// TwinCAT 3 PLC project SSP_M
// ProgramVersion: 3.1.4024.0
// libraries:
//   EfficientIO Communicator, * (EfficientIO)
//   EfficientIO Energy Basic, * (EfficientIO)
//   EfficientIO ModbusTCP, * (EfficientIO)
//   Lynus Persistent Data V1, * (Lynus AG)
//   Lynus Standards, * (EfficientIO)
//   Tc2_EtherCAT, * (Beckhoff Automation GmbH)
//   Tc2_Standard, * (Beckhoff Automation GmbH)
//   Tc2_System, * (Beckhoff Automation GmbH)
//   Tc2_Utilities, * (Beckhoff Automation GmbH)
//   Tc3_Module, * (Beckhoff Automation GmbH)
// project tree:
//   / FastTask.TcTTO, PlcTask.TcTTO, SlowTask.TcTTO (not stored)
//   FBs/EL3443_DPM/DUTs/ E_EL3443_DPM_Phase.TcDUT (not stored), E_EL3443_DPM_Total.TcDUT (not stored), MDP5001_341_7CD731EE.TcDUT (not stored), MDP5001_341_I_7CD731EE.TcDUT (not stored), MDP5001_341_O_7CD731EE.TcDUT (not stored), ST_EL3443_DPM_MUX_REAL.TcDUT (not stored), ST_EL3443_DPM_MUX_ULINT.TcDUT (not stored), ST_EL3443_DPM_StatusLx.TcDUT (not stored), ST_EL3443_DPM_StatusTotal.TcDUT (not stored), ST_EL3443_DPM_VariantLx.TcDUT (not stored), ST_EL3443_DPM_VariantTotal.TcDUT (not stored), ST_EL3443_DPM_VariantValues.TcDUT (not stored)
//   FBs/EL3443_DPM/ FB_EL3443_DPM.TcPOU (not stored)
//   FBs/EL3446 FW02 or higher/DUTs/ E_EL3446_Phase.TcDUT (not stored), MDP5001_342_066CA8C6.TcDUT (not stored), MDP5001_342_I_066CA8C6.TcDUT (not stored), MDP5001_342_O_066CA8C6.TcDUT, ST_EL3446_MUX_REAL.TcDUT (not stored), ST_EL3446_MUX_ULINT.TcDUT (not stored), ST_EL3446_StatusIx.TcDUT (not stored), ST_EL3446_VariantIx.TcDUT (not stored), ST_EL3446_VariantValues.TcDUT (not stored)
//   FBs/EL3446 FW02 or higher/ FB_EL3446.TcPOU (not stored)
//   FBs/ FB_CoE_EL3443.TcPOU (not stored), FB_CoE_EL3446.TcPOU (not stored), FB_EM_Beckhoff_EL3443.TcPOU (not stored), FB_EM_Beckhoff_EL3446.TcPOU (not stored)
//   POUs/ prgComEffIO.TcPOU, prgEM.TcPOU, prgEMS.TcPOU, prgHW.TcPOU, prgModbus.TcPOU, prgPersistent.TcPOU, prgRWEffIO.TcPOU (not stored), prgVarEffIO.TcPOU (not stored)
// real-time tasks:
//   TASK MiddleTask: cycle T#10ms, priority 20, ADS port 350
//   TASK FastTask: cycle T#5ms, priority 19, ADS port 351
//   TASK SlowTask: cycle T#20ms, priority 21, ADS port 352
// I/O:
//   DEVICE Device 1 (Beckhoff CCAT)
//   DEVICE Device 2 (EtherCAT), AmsNetId 5.146.126.209.3.1
//     Term 1 (EK1200) [EK1200-5000 EtherCAT Power supply (2A E-Bus)]
//       Term 6 (EL3443) [EL3443 3Ch. Power Measuring]
//       Term 2 (EL3443) [EL3443 3Ch. Power Measuring]
//       Term 3 (EL3446) [EL3446 6 Ch.DPM Current Measurement Terminal]
//       Term 4 (EL3446) [EL3446 6 Ch.DPM Current Measurement Terminal]
//       Term 5 (EL9011) [EL9011 End Terminal]
//   DEVICE Gerät 3 (RT-Ethernet Protocol), AmsNetId 5.146.126.209.4.1
//     BK9050 (BK9050-0000 192.168.1.235)
// variable links:
//   SSP-M/SSP-M Instance <-> Device 2 (EtherCAT)/Term 1 (EK1200)/Term 2 (EL3443)
//     PlcTask Inputs/prgHW.MDP5001_342_DPM_Data_Data_{1..20} <-> DPM Data/Data {1..20}  (20 links)
//     PlcTask Inputs/prgHW.MDP5001_342_L1_Basic_Current <-> L1 Basic/Current
//     PlcTask Inputs/prgHW.MDP5001_342_L2_Basic_Current <-> L2 Basic/Current
//     PlcTask Inputs/prgHW.MDP5001_342_L3_Basic_Current <-> L3 Basic/Current
//     PlcTask Inputs/prgHW.MDP5001_342_L1_Basic_Voltage <-> L1 Basic/Voltage
//     PlcTask Inputs/prgHW.MDP5001_342_L2_Basic_Voltage <-> L2 Basic/Voltage
//     PlcTask Inputs/prgHW.MDP5001_342_L3_Basic_Voltage <-> L3 Basic/Voltage
//     PlcTask Inputs/prgHW.MDP5001_342_L1_Power_Active_Power <-> L1 Power/Active Power
//     PlcTask Inputs/prgHW.MDP5001_342_L2_Power_Active_Power <-> L2 Power/Active Power
//     PlcTask Inputs/prgHW.MDP5001_342_L3_Power_Active_Power <-> L3 Power/Active Power
//     PlcTask Inputs/prgHW.MDP5001_342_L1_Power_Apparent_Power <-> L1 Power/Apparent Power
//     PlcTask Inputs/prgHW.MDP5001_342_L2_Power_Apparent_Power <-> L2 Power/Apparent Power
//     PlcTask Inputs/prgHW.MDP5001_342_L3_Power_Apparent_Power <-> L3 Power/Apparent Power
//     PlcTask Inputs/prgHW.MDP5001_342_L1_Power_Power_Factor <-> L1 Power/Power Factor
//     PlcTask Inputs/prgHW.MDP5001_342_L2_Power_Power_Factor <-> L2 Power/Power Factor
//     PlcTask Inputs/prgHW.MDP5001_342_L3_Power_Power_Factor <-> L3 Power/Power Factor
//     PlcTask Inputs/prgHW.MDP5001_342_L1_Power_Reactive_Power <-> L1 Power/Reactive Power
//     PlcTask Inputs/prgHW.MDP5001_342_L2_Power_Reactive_Power <-> L2 Power/Reactive Power
//     PlcTask Inputs/prgHW.MDP5001_342_L3_Power_Reactive_Power <-> L3 Power/Reactive Power
//     PlcTask Inputs/prgHW.MDP5001_342_L1_Status_Current_Guard_Error <-> L1 Status/Current Guard Error
//     PlcTask Inputs/prgHW.MDP5001_342_L2_Status_Current_Guard_Error <-> L2 Status/Current Guard Error
//     PlcTask Inputs/prgHW.MDP5001_342_L3_Status_Current_Guard_Error <-> L3 Status/Current Guard Error
//     PlcTask Inputs/prgHW.MDP5001_342_L1_Status_Current_Guard_Warning <-> L1 Status/Current Guard Warning
//     PlcTask Inputs/prgHW.MDP5001_342_L2_Status_Current_Guard_Warning <-> L2 Status/Current Guard Warning
//     PlcTask Inputs/prgHW.MDP5001_342_L3_Status_Current_Guard_Warning <-> L3 Status/Current Guard Warning
//     PlcTask Inputs/prgHW.MDP5001_342_L1_Status_Inaccurate_Current <-> L1 Status/Inaccurate Current
//     PlcTask Inputs/prgHW.MDP5001_342_L2_Status_Inaccurate_Current <-> L2 Status/Inaccurate Current
//     PlcTask Inputs/prgHW.MDP5001_342_L3_Status_Inaccurate_Current <-> L3 Status/Inaccurate Current
//     PlcTask Inputs/prgHW.MDP5001_342_L1_Status_Inaccurate_Voltage <-> L1 Status/Inaccurate Voltage
//     PlcTask Inputs/prgHW.MDP5001_342_L2_Status_Inaccurate_Voltage <-> L2 Status/Inaccurate Voltage
//     PlcTask Inputs/prgHW.MDP5001_342_L3_Status_Inaccurate_Voltage <-> L3 Status/Inaccurate Voltage
//     PlcTask Inputs/prgHW.MDP5001_342_L1_Status_Overcurrent <-> L1 Status/Overcurrent
//     PlcTask Inputs/prgHW.MDP5001_342_L2_Status_Overcurrent <-> L2 Status/Overcurrent
//     PlcTask Inputs/prgHW.MDP5001_342_L3_Status_Overcurrent <-> L3 Status/Overcurrent
//     PlcTask Inputs/prgHW.MDP5001_342_L1_Status_Overvoltage <-> L1 Status/Overvoltage
//     PlcTask Inputs/prgHW.MDP5001_342_L2_Status_Overvoltage <-> L2 Status/Overvoltage
//     PlcTask Inputs/prgHW.MDP5001_342_L3_Status_Overvoltage <-> L3 Status/Overvoltage
//     PlcTask Inputs/prgHW.MDP5001_342_L1_Status_TxPDO_Toggle <-> L1 Status/TxPDO Toggle
//     PlcTask Inputs/prgHW.MDP5001_342_L2_Status_TxPDO_Toggle <-> L2 Status/TxPDO Toggle
//     PlcTask Inputs/prgHW.MDP5001_342_L3_Status_TxPDO_Toggle <-> L3 Status/TxPDO Toggle
//     PlcTask Inputs/prgHW.MDP5001_342_L1_Status_Voltage_Guard_Error <-> L1 Status/Voltage Guard Error
//     PlcTask Inputs/prgHW.MDP5001_342_L2_Status_Voltage_Guard_Error <-> L2 Status/Voltage Guard Error
//     PlcTask Inputs/prgHW.MDP5001_342_L3_Status_Voltage_Guard_Error <-> L3 Status/Voltage Guard Error
//     PlcTask Inputs/prgHW.MDP5001_342_L1_Status_Voltage_Guard_Warning <-> L1 Status/Voltage Guard Warning
//     PlcTask Inputs/prgHW.MDP5001_342_L2_Status_Voltage_Guard_Warning <-> L2 Status/Voltage Guard Warning
//     PlcTask Inputs/prgHW.MDP5001_342_L3_Status_Voltage_Guard_Warning <-> L3 Status/Voltage Guard Warning
//     PlcTask Inputs/prgHW.MDP5001_342_L1_Status_Voltage_Sign_Bit <-> L1 Status/Voltage Sign Bit
//     PlcTask Inputs/prgHW.MDP5001_342_L2_Status_Voltage_Sign_Bit <-> L2 Status/Voltage Sign Bit
//     PlcTask Inputs/prgHW.MDP5001_342_L3_Status_Voltage_Sign_Bit <-> L3 Status/Voltage Sign Bit
//     PlcTask Inputs/prgHW.MDP5001_342_Total_Basic_Calculated_Neutral_Line_Current <-> Total Basic/Calculated Neutral Line Current
//     PlcTask Inputs/prgHW.MDP5001_342_Total_Basic_Frequency <-> Total Basic/Frequency
//     PlcTask Inputs/prgHW.MDP5001_342_Total_Basic_Power_Factor <-> Total Basic/Power Factor
//     PlcTask Inputs/prgHW.MDP5001_342_Total_Status_Active_Power_Guard_Error <-> Total Status/Active Power Guard Error
//     PlcTask Inputs/prgHW.MDP5001_342_Total_Status_Active_Power_Guard_Warning <-> Total Status/Active Power Guard Warning
//     PlcTask Inputs/prgHW.MDP5001_342_Total_Status_Apparent_Power_Guard_Error <-> Total Status/Apparent Power Guard Error
//     PlcTask Inputs/prgHW.MDP5001_342_Total_Status_Apparent_Power_Guard_Warning <-> Total Status/Apparent Power Guard Warning
//     PlcTask Inputs/prgHW.MDP5001_342_Total_Status_Frequency_Guard_Error <-> Total Status/Frequency Guard Error
//     PlcTask Inputs/prgHW.MDP5001_342_Total_Status_Frequency_Guard_Warning <-> Total Status/Frequency Guard Warning
//     PlcTask Inputs/prgHW.MDP5001_342_Total_Status_Grid_Direction <-> Total Status/Grid Direction
//     PlcTask Inputs/prgHW.MDP5001_342_Total_Status_Neutral_Current_Guard_Error <-> Total Status/Neutral Current Guard Error
//     PlcTask Inputs/prgHW.MDP5001_342_Total_Status_Neutral_Current_Guard_Warning <-> Total Status/Neutral Current Guard Warning
//     PlcTask Inputs/prgHW.MDP5001_342_Total_Status_Power_Quality_Factor <-> Total Status/Power Quality Factor
//     PlcTask Inputs/prgHW.MDP5001_342_Total_Status_Power_Quality_Guard_Error <-> Total Status/Power Quality Guard Error
//     PlcTask Inputs/prgHW.MDP5001_342_Total_Status_Power_Quality_Guard_Warning <-> Total Status/Power Quality Guard Warning
//     PlcTask Inputs/prgHW.MDP5001_342_Total_Status_System_State <-> Total Status/System State
//     PlcTask Inputs/prgHW.MDP5001_342_Total_Status_TxPDO_State <-> Total Status/TxPDO State
//     PlcTask Inputs/prgHW.MDP5001_342_Total_Status_TxPDO_Toggle <-> Total Status/TxPDO Toggle
//     PlcTask Inputs/prgHW.MDP5001_342_Total_Variant_Value_In_Index_1_REAL <-> Total Variant Value In/Index 1 REAL
//     PlcTask Inputs/prgHW.MDP5001_342_Total_Variant_Value_In_Index_2_REAL <-> Total Variant Value In/Index 2 REAL
//     PlcTask Inputs/prgHW.MDP5001_342_Total_Variant_Value_In_Index_3_REAL <-> Total Variant Value In/Index 3 REAL
//     PlcTask Inputs/prgHW.MDP5001_342_Total_Variant_Value_In_Index_4_ULINT <-> Total Variant Value In/Index 4 ULINT
//     PlcTask Inputs/prgHW.MDP5001_342_Total_Variant_Value_In_TxPDO_Toggle <-> Total Variant Value In/TxPDO Toggle
//     PlcTask Inputs/prgHW.MDP5001_342_Total_Variant_Value_In_Value_1_REAL <-> Total Variant Value In/Value 1 REAL
//     PlcTask Inputs/prgHW.MDP5001_342_Total_Variant_Value_In_Value_2_REAL <-> Total Variant Value In/Value 2 REAL
//     PlcTask Inputs/prgHW.MDP5001_342_Total_Variant_Value_In_Value_3_REAL <-> Total Variant Value In/Value 3 REAL
//     PlcTask Inputs/prgHW.MDP5001_342_Total_Variant_Value_In_Value_4_ULINT <-> Total Variant Value In/Value 4 ULINT
//     PlcTask Outputs/prgHW.MDP5001_342_Total_Interval_Reset_Interval <-> Total Interval/Reset Interval
//     PlcTask Outputs/prgHW.MDP5001_342_Total_Variant_Value_Out_Index_1_REAL <-> Total Variant Value Out/Index 1 REAL
//     PlcTask Outputs/prgHW.MDP5001_342_Total_Variant_Value_Out_Index_2_REAL <-> Total Variant Value Out/Index 2 REAL
//     PlcTask Outputs/prgHW.MDP5001_342_Total_Variant_Value_Out_Index_3_REAL <-> Total Variant Value Out/Index 3 REAL
//     PlcTask Outputs/prgHW.MDP5001_342_Total_Variant_Value_Out_Index_4_ULINT <-> Total Variant Value Out/Index 4 ULINT
//   SSP-M/SSP-M Instance <-> Device 2 (EtherCAT)/Term 1 (EK1200)/Term 3 (EL3446)
//     PlcTask Inputs/prgHW.MDP5001_342_DPM_Variant_Value_In_Index_1_REAL_1 <-> DPM Variant Value In/Index 1 REAL
//     PlcTask Inputs/prgHW.MDP5001_342_DPM_Variant_Value_In_Index_2_REAL_1 <-> DPM Variant Value In/Index 2 REAL
//     PlcTask Inputs/prgHW.MDP5001_342_DPM_Variant_Value_In_Index_3_REAL_1 <-> DPM Variant Value In/Index 3 REAL
//     PlcTask Inputs/prgHW.MDP5001_342_DPM_Variant_Value_In_Index_4_ULINT_1 <-> DPM Variant Value In/Index 4 ULINT
//     PlcTask Inputs/prgHW.MDP5001_342_DPM_Variant_Value_In_TxPDO_Toggle_1 <-> DPM Variant Value In/TxPDO Toggle
//     PlcTask Inputs/prgHW.MDP5001_342_DPM_Variant_Value_In_Value_1_REAL_1 <-> DPM Variant Value In/Value 1 REAL
//     PlcTask Inputs/prgHW.MDP5001_342_DPM_Variant_Value_In_Value_2_REAL_1 <-> DPM Variant Value In/Value 2 REAL
//     PlcTask Inputs/prgHW.MDP5001_342_DPM_Variant_Value_In_Value_3_REAL_1 <-> DPM Variant Value In/Value 3 REAL
//     PlcTask Inputs/prgHW.MDP5001_342_DPM_Variant_Value_In_Value_4_ULINT_1 <-> DPM Variant Value In/Value 4 ULINT
//     PlcTask Inputs/prgHW.MDP5001_342_I{1..6}_Channel_Active_Energy_1 <-> I{1..6} Channel/Active Energy  (6 links)
//     PlcTask Inputs/prgHW.MDP5001_342_I{1..6}_Channel_Active_Power_1 <-> I{1..6} Channel/Active Power  (6 links)
//     PlcTask Inputs/prgHW.MDP5001_342_I{1..6}_Channel_Active_Power_Guard_Error_1 <-> I{1..6} Channel/Active Power Guard Error  (6 links)
//     PlcTask Inputs/prgHW.MDP5001_342_I{1..6}_Channel_Active_Power_Guard_Warning_1 <-> I{1..6} Channel/Active Power Guard Warning  (6 links)
//     PlcTask Inputs/prgHW.MDP5001_342_I{1..6}_Channel_Apparent_Power_1 <-> I{1..6} Channel/Apparent Power  (6 links)
//     PlcTask Inputs/prgHW.MDP5001_342_I{1..6}_Channel_Apparent_Power_Guard_Error_1 <-> I{1..6} Channel/Apparent Power Guard Error  (6 links)
//     PlcTask Inputs/prgHW.MDP5001_342_I{1..6}_Channel_Apparent_Power_Guard_Warning_1 <-> I{1..6} Channel/Apparent Power Guard Warning  (6 links)
//     PlcTask Inputs/prgHW.MDP5001_342_I{1..6}_Channel_Current_1 <-> I{1..6} Channel/Current  (6 links)
//     PlcTask Inputs/prgHW.MDP5001_342_I{1..6}_Channel_Current_Guard_Error_1 <-> I{1..6} Channel/Current Guard Error  (6 links)
//     PlcTask Inputs/prgHW.MDP5001_342_I{1..6}_Channel_Current_Guard_Warning_1 <-> I{1..6} Channel/Current Guard Warning  (6 links)
//     PlcTask Inputs/prgHW.MDP5001_342_I{1..6}_Channel_DPM_Inaccurate_1 <-> I{1..6} Channel/DPM Inaccurate  (6 links)
//     PlcTask Inputs/prgHW.MDP5001_342_I{1..6}_Channel_DPM_Timeout_1 <-> I{1..6} Channel/DPM Timeout  (6 links)
//     PlcTask Inputs/prgHW.MDP5001_342_I{1..6}_Channel_Inaccurate_Current_1 <-> I{1..6} Channel/Inaccurate Current  (6 links)
//     PlcTask Inputs/prgHW.MDP5001_342_I{1..6}_Channel_Overcurrent_1 <-> I{1..6} Channel/Overcurrent  (6 links)
//     PlcTask Inputs/prgHW.MDP5001_342_I{1..6}_Channel_Reactive_Power_Fundamental_1 <-> I{1..6} Channel/Reactive Power Fundamental  (6 links)
//     PlcTask Inputs/prgHW.MDP5001_342_I{1..6}_Channel_Reactive_Power_Guard_Error_1 <-> I{1..6} Channel/Reactive Power Guard Error  (6 links)
//     PlcTask Inputs/prgHW.MDP5001_342_I{1..6}_Channel_Reactive_Power_Guard_Warning_1 <-> I{1..6} Channel/Reactive Power Guard Warning  (6 links)
//     PlcTask Inputs/prgHW.MDP5001_342_I{1..6}_Channel_TxPDO_Toggle_1 <-> I{1..6} Channel/TxPDO Toggle  (6 links)
//     PlcTask Outputs/prgHW.MDP5001_342_DPM_Data_Data_{1..20}_1 <-> DPM Data/Data {1..20}  (20 links)
//     PlcTask Outputs/prgHW.MDP5001_342_DPM_Variant_Value_Out_Index_1_REAL_1 <-> DPM Variant Value Out/Index 1 REAL
//     PlcTask Outputs/prgHW.MDP5001_342_DPM_Variant_Value_Out_Index_2_REAL_1 <-> DPM Variant Value Out/Index 2 REAL
//     PlcTask Outputs/prgHW.MDP5001_342_DPM_Variant_Value_Out_Index_3_REAL_1 <-> DPM Variant Value Out/Index 3 REAL
//     PlcTask Outputs/prgHW.MDP5001_342_DPM_Variant_Value_Out_Index_4_ULINT_1 <-> DPM Variant Value Out/Index 4 ULINT
//   SSP-M/SSP-M Instance <-> Device 2 (EtherCAT)/Term 1 (EK1200)/Term 4 (EL3446)
//     PlcTask Inputs/prgHW.MDP5001_342_DPM_Variant_Value_In_Index_1_REAL_2 <-> DPM Variant Value In/Index 1 REAL
//     PlcTask Inputs/prgHW.MDP5001_342_DPM_Variant_Value_In_Index_2_REAL_2 <-> DPM Variant Value In/Index 2 REAL
//     PlcTask Inputs/prgHW.MDP5001_342_DPM_Variant_Value_In_Index_3_REAL_2 <-> DPM Variant Value In/Index 3 REAL
//     PlcTask Inputs/prgHW.MDP5001_342_DPM_Variant_Value_In_Index_4_ULINT_2 <-> DPM Variant Value In/Index 4 ULINT
//     PlcTask Inputs/prgHW.MDP5001_342_DPM_Variant_Value_In_TxPDO_Toggle_2 <-> DPM Variant Value In/TxPDO Toggle
//     PlcTask Inputs/prgHW.MDP5001_342_DPM_Variant_Value_In_Value_1_REAL_2 <-> DPM Variant Value In/Value 1 REAL
//     PlcTask Inputs/prgHW.MDP5001_342_DPM_Variant_Value_In_Value_2_REAL_2 <-> DPM Variant Value In/Value 2 REAL
//     PlcTask Inputs/prgHW.MDP5001_342_DPM_Variant_Value_In_Value_3_REAL_2 <-> DPM Variant Value In/Value 3 REAL
//     PlcTask Inputs/prgHW.MDP5001_342_DPM_Variant_Value_In_Value_4_ULINT_2 <-> DPM Variant Value In/Value 4 ULINT
//     PlcTask Inputs/prgHW.MDP5001_342_I{1..6}_Channel_Active_Energy_2 <-> I{1..6} Channel/Active Energy  (6 links)
//     PlcTask Inputs/prgHW.MDP5001_342_I{1..6}_Channel_Active_Power_2 <-> I{1..6} Channel/Active Power  (6 links)
//     PlcTask Inputs/prgHW.MDP5001_342_I{1..6}_Channel_Active_Power_Guard_Error_2 <-> I{1..6} Channel/Active Power Guard Error  (6 links)
//     PlcTask Inputs/prgHW.MDP5001_342_I{1..6}_Channel_Active_Power_Guard_Warning_2 <-> I{1..6} Channel/Active Power Guard Warning  (6 links)
//     PlcTask Inputs/prgHW.MDP5001_342_I{1..6}_Channel_Apparent_Power_2 <-> I{1..6} Channel/Apparent Power  (6 links)
//     PlcTask Inputs/prgHW.MDP5001_342_I{1..6}_Channel_Apparent_Power_Guard_Error_2 <-> I{1..6} Channel/Apparent Power Guard Error  (6 links)
//     PlcTask Inputs/prgHW.MDP5001_342_I{1..6}_Channel_Apparent_Power_Guard_Warning_2 <-> I{1..6} Channel/Apparent Power Guard Warning  (6 links)
//     PlcTask Inputs/prgHW.MDP5001_342_I{1..6}_Channel_Current_2 <-> I{1..6} Channel/Current  (6 links)
//     PlcTask Inputs/prgHW.MDP5001_342_I{1..6}_Channel_Current_Guard_Error_2 <-> I{1..6} Channel/Current Guard Error  (6 links)
//     PlcTask Inputs/prgHW.MDP5001_342_I{1..6}_Channel_Current_Guard_Warning_2 <-> I{1..6} Channel/Current Guard Warning  (6 links)
//     PlcTask Inputs/prgHW.MDP5001_342_I{1..6}_Channel_DPM_Inaccurate_2 <-> I{1..6} Channel/DPM Inaccurate  (6 links)
//     PlcTask Inputs/prgHW.MDP5001_342_I{1..6}_Channel_DPM_Timeout_2 <-> I{1..6} Channel/DPM Timeout  (6 links)
//     PlcTask Inputs/prgHW.MDP5001_342_I{1..6}_Channel_Inaccurate_Current_2 <-> I{1..6} Channel/Inaccurate Current  (6 links)
//     PlcTask Inputs/prgHW.MDP5001_342_I{1..6}_Channel_Overcurrent_2 <-> I{1..6} Channel/Overcurrent  (6 links)
//     PlcTask Inputs/prgHW.MDP5001_342_I{1..6}_Channel_Reactive_Power_Fundamental_2 <-> I{1..6} Channel/Reactive Power Fundamental  (6 links)
//     PlcTask Inputs/prgHW.MDP5001_342_I{1..6}_Channel_Reactive_Power_Guard_Error_2 <-> I{1..6} Channel/Reactive Power Guard Error  (6 links)
//     PlcTask Inputs/prgHW.MDP5001_342_I{1..6}_Channel_Reactive_Power_Guard_Warning_2 <-> I{1..6} Channel/Reactive Power Guard Warning  (6 links)
//     PlcTask Inputs/prgHW.MDP5001_342_I{1..6}_Channel_TxPDO_Toggle_2 <-> I{1..6} Channel/TxPDO Toggle  (6 links)
//     PlcTask Outputs/prgHW.MDP5001_342_DPM_Data_Data_{1..20}_2 <-> DPM Data/Data {1..20}  (20 links)
//     PlcTask Outputs/prgHW.MDP5001_342_DPM_Variant_Value_Out_Index_1_REAL_2 <-> DPM Variant Value Out/Index 1 REAL
//     PlcTask Outputs/prgHW.MDP5001_342_DPM_Variant_Value_Out_Index_2_REAL_2 <-> DPM Variant Value Out/Index 2 REAL
//     PlcTask Outputs/prgHW.MDP5001_342_DPM_Variant_Value_Out_Index_3_REAL_2 <-> DPM Variant Value Out/Index 3 REAL
//     PlcTask Outputs/prgHW.MDP5001_342_DPM_Variant_Value_Out_Index_4_ULINT_2 <-> DPM Variant Value Out/Index 4 ULINT
//   SSP-M/SSP-M Instance <-> Device 2 (EtherCAT)/Term 1 (EK1200)/Term 6 (EL3443)
//     PlcTask Inputs/prgHW.MDP5001_341_DPM_Data_Data_{1..20} <-> DPM Data/Data {1..20}  (20 links)
//     PlcTask Inputs/prgHW.MDP5001_341_L1_Basic_Current <-> L1 Basic/Current
//     PlcTask Inputs/prgHW.MDP5001_341_L2_Basic_Current <-> L2 Basic/Current
//     PlcTask Inputs/prgHW.MDP5001_341_L3_Basic_Current <-> L3 Basic/Current
//     PlcTask Inputs/prgHW.MDP5001_341_L1_Basic_Voltage <-> L1 Basic/Voltage
//     PlcTask Inputs/prgHW.MDP5001_341_L2_Basic_Voltage <-> L2 Basic/Voltage
//     PlcTask Inputs/prgHW.MDP5001_341_L3_Basic_Voltage <-> L3 Basic/Voltage
//     PlcTask Inputs/prgHW.MDP5001_341_L1_Power_Active_Power <-> L1 Power/Active Power
//     PlcTask Inputs/prgHW.MDP5001_341_L2_Power_Active_Power <-> L2 Power/Active Power
//     PlcTask Inputs/prgHW.MDP5001_341_L3_Power_Active_Power <-> L3 Power/Active Power
//     PlcTask Inputs/prgHW.MDP5001_341_L1_Power_Apparent_Power <-> L1 Power/Apparent Power
//     PlcTask Inputs/prgHW.MDP5001_341_L2_Power_Apparent_Power <-> L2 Power/Apparent Power
//     PlcTask Inputs/prgHW.MDP5001_341_L3_Power_Apparent_Power <-> L3 Power/Apparent Power
//     PlcTask Inputs/prgHW.MDP5001_341_L1_Power_Power_Factor <-> L1 Power/Power Factor
//     PlcTask Inputs/prgHW.MDP5001_341_L2_Power_Power_Factor <-> L2 Power/Power Factor
//     PlcTask Inputs/prgHW.MDP5001_341_L3_Power_Power_Factor <-> L3 Power/Power Factor
//     PlcTask Inputs/prgHW.MDP5001_341_L1_Power_Reactive_Power <-> L1 Power/Reactive Power
//     PlcTask Inputs/prgHW.MDP5001_341_L2_Power_Reactive_Power <-> L2 Power/Reactive Power
//     PlcTask Inputs/prgHW.MDP5001_341_L3_Power_Reactive_Power <-> L3 Power/Reactive Power
//     PlcTask Inputs/prgHW.MDP5001_341_L1_Status_Current_Guard_Error <-> L1 Status/Current Guard Error
//     PlcTask Inputs/prgHW.MDP5001_341_L2_Status_Current_Guard_Error <-> L2 Status/Current Guard Error
//     PlcTask Inputs/prgHW.MDP5001_341_L3_Status_Current_Guard_Error <-> L3 Status/Current Guard Error
//     PlcTask Inputs/prgHW.MDP5001_341_L1_Status_Current_Guard_Warning <-> L1 Status/Current Guard Warning
//     PlcTask Inputs/prgHW.MDP5001_341_L2_Status_Current_Guard_Warning <-> L2 Status/Current Guard Warning
//     PlcTask Inputs/prgHW.MDP5001_341_L3_Status_Current_Guard_Warning <-> L3 Status/Current Guard Warning
//     PlcTask Inputs/prgHW.MDP5001_341_L1_Status_Inaccurate_Current <-> L1 Status/Inaccurate Current
//     PlcTask Inputs/prgHW.MDP5001_341_L2_Status_Inaccurate_Current <-> L2 Status/Inaccurate Current
//     PlcTask Inputs/prgHW.MDP5001_341_L3_Status_Inaccurate_Current <-> L3 Status/Inaccurate Current
//     PlcTask Inputs/prgHW.MDP5001_341_L1_Status_Inaccurate_Voltage <-> L1 Status/Inaccurate Voltage
//     PlcTask Inputs/prgHW.MDP5001_341_L2_Status_Inaccurate_Voltage <-> L2 Status/Inaccurate Voltage
//     PlcTask Inputs/prgHW.MDP5001_341_L3_Status_Inaccurate_Voltage <-> L3 Status/Inaccurate Voltage
//     PlcTask Inputs/prgHW.MDP5001_341_L1_Status_Overcurrent <-> L1 Status/Overcurrent
//     PlcTask Inputs/prgHW.MDP5001_341_L2_Status_Overcurrent <-> L2 Status/Overcurrent
//     PlcTask Inputs/prgHW.MDP5001_341_L3_Status_Overcurrent <-> L3 Status/Overcurrent
//     PlcTask Inputs/prgHW.MDP5001_341_L1_Status_Overvoltage <-> L1 Status/Overvoltage
//     PlcTask Inputs/prgHW.MDP5001_341_L2_Status_Overvoltage <-> L2 Status/Overvoltage
//     PlcTask Inputs/prgHW.MDP5001_341_L3_Status_Overvoltage <-> L3 Status/Overvoltage
//     PlcTask Inputs/prgHW.MDP5001_341_L1_Status_TxPDO_Toggle <-> L1 Status/TxPDO Toggle
//     PlcTask Inputs/prgHW.MDP5001_341_L2_Status_TxPDO_Toggle <-> L2 Status/TxPDO Toggle
//     PlcTask Inputs/prgHW.MDP5001_341_L3_Status_TxPDO_Toggle <-> L3 Status/TxPDO Toggle
//     PlcTask Inputs/prgHW.MDP5001_341_L1_Status_Voltage_Guard_Error <-> L1 Status/Voltage Guard Error
//     PlcTask Inputs/prgHW.MDP5001_341_L2_Status_Voltage_Guard_Error <-> L2 Status/Voltage Guard Error
//     PlcTask Inputs/prgHW.MDP5001_341_L3_Status_Voltage_Guard_Error <-> L3 Status/Voltage Guard Error
//     PlcTask Inputs/prgHW.MDP5001_341_L1_Status_Voltage_Guard_Warning <-> L1 Status/Voltage Guard Warning
//     PlcTask Inputs/prgHW.MDP5001_341_L2_Status_Voltage_Guard_Warning <-> L2 Status/Voltage Guard Warning
//     PlcTask Inputs/prgHW.MDP5001_341_L3_Status_Voltage_Guard_Warning <-> L3 Status/Voltage Guard Warning
//     PlcTask Inputs/prgHW.MDP5001_341_L1_Status_Voltage_Sign_Bit <-> L1 Status/Voltage Sign Bit
//     PlcTask Inputs/prgHW.MDP5001_341_L2_Status_Voltage_Sign_Bit <-> L2 Status/Voltage Sign Bit
//     PlcTask Inputs/prgHW.MDP5001_341_L3_Status_Voltage_Sign_Bit <-> L3 Status/Voltage Sign Bit
//     PlcTask Inputs/prgHW.MDP5001_341_Total_Basic_Calculated_Neutral_Line_Current <-> Total Basic/Calculated Neutral Line Current
//     PlcTask Inputs/prgHW.MDP5001_341_Total_Basic_Frequency <-> Total Basic/Frequency
//     PlcTask Inputs/prgHW.MDP5001_341_Total_Basic_Power_Factor <-> Total Basic/Power Factor
//     PlcTask Inputs/prgHW.MDP5001_341_Total_Status_Active_Power_Guard_Error <-> Total Status/Active Power Guard Error
//     PlcTask Inputs/prgHW.MDP5001_341_Total_Status_Active_Power_Guard_Warning <-> Total Status/Active Power Guard Warning
//     PlcTask Inputs/prgHW.MDP5001_341_Total_Status_Apparent_Power_Guard_Error <-> Total Status/Apparent Power Guard Error
//     PlcTask Inputs/prgHW.MDP5001_341_Total_Status_Apparent_Power_Guard_Warning <-> Total Status/Apparent Power Guard Warning
//     PlcTask Inputs/prgHW.MDP5001_341_Total_Status_Frequency_Guard_Error <-> Total Status/Frequency Guard Error
//     PlcTask Inputs/prgHW.MDP5001_341_Total_Status_Frequency_Guard_Warning <-> Total Status/Frequency Guard Warning
//     PlcTask Inputs/prgHW.MDP5001_341_Total_Status_Grid_Direction <-> Total Status/Grid Direction
//     PlcTask Inputs/prgHW.MDP5001_341_Total_Status_Neutral_Current_Guard_Error <-> Total Status/Neutral Current Guard Error
//     PlcTask Inputs/prgHW.MDP5001_341_Total_Status_Neutral_Current_Guard_Warning <-> Total Status/Neutral Current Guard Warning
//     PlcTask Inputs/prgHW.MDP5001_341_Total_Status_Power_Quality_Factor <-> Total Status/Power Quality Factor
//     PlcTask Inputs/prgHW.MDP5001_341_Total_Status_Power_Quality_Guard_Error <-> Total Status/Power Quality Guard Error
//     PlcTask Inputs/prgHW.MDP5001_341_Total_Status_Power_Quality_Guard_Warning <-> Total Status/Power Quality Guard Warning
//     PlcTask Inputs/prgHW.MDP5001_341_Total_Status_System_State <-> Total Status/System State
//     PlcTask Inputs/prgHW.MDP5001_341_Total_Status_TxPDO_State <-> Total Status/TxPDO State
//     PlcTask Inputs/prgHW.MDP5001_341_Total_Status_TxPDO_Toggle <-> Total Status/TxPDO Toggle
//     PlcTask Inputs/prgHW.MDP5001_341_Total_Variant_Value_In_Index_1_REAL <-> Total Variant Value In/Index 1 REAL
//     PlcTask Inputs/prgHW.MDP5001_341_Total_Variant_Value_In_Index_2_REAL <-> Total Variant Value In/Index 2 REAL
//     PlcTask Inputs/prgHW.MDP5001_341_Total_Variant_Value_In_Index_3_REAL <-> Total Variant Value In/Index 3 REAL
//     PlcTask Inputs/prgHW.MDP5001_341_Total_Variant_Value_In_Index_4_ULINT <-> Total Variant Value In/Index 4 ULINT
//     PlcTask Inputs/prgHW.MDP5001_341_Total_Variant_Value_In_TxPDO_Toggle <-> Total Variant Value In/TxPDO Toggle
//     PlcTask Inputs/prgHW.MDP5001_341_Total_Variant_Value_In_Value_1_REAL <-> Total Variant Value In/Value 1 REAL
//     PlcTask Inputs/prgHW.MDP5001_341_Total_Variant_Value_In_Value_2_REAL <-> Total Variant Value In/Value 2 REAL
//     PlcTask Inputs/prgHW.MDP5001_341_Total_Variant_Value_In_Value_3_REAL <-> Total Variant Value In/Value 3 REAL
//     PlcTask Inputs/prgHW.MDP5001_341_Total_Variant_Value_In_Value_4_ULINT <-> Total Variant Value In/Value 4 ULINT
//     PlcTask Outputs/prgHW.MDP5001_341_Total_Interval_Reset_Interval <-> Total Interval/Reset Interval
//     PlcTask Outputs/prgHW.MDP5001_341_Total_Variant_Value_Out_Index_1_REAL <-> Total Variant Value Out/Index 1 REAL
//     PlcTask Outputs/prgHW.MDP5001_341_Total_Variant_Value_Out_Index_2_REAL <-> Total Variant Value Out/Index 2 REAL
//     PlcTask Outputs/prgHW.MDP5001_341_Total_Variant_Value_Out_Index_3_REAL <-> Total Variant Value Out/Index 3 REAL
//     PlcTask Outputs/prgHW.MDP5001_341_Total_Variant_Value_Out_Index_4_ULINT <-> Total Variant Value Out/Index 4 ULINT
//   SSP-M/SSP-M Instance <-> Device 3 (RT-Ethernet Protocol)/BK9050 (BK9050-0000 192.168.1.235)
//     PlcTask Inputs/prgEM.fb_KL3403.fbKL3403.byStateCH1 <-> Term 2 (KL3403)/Channel 1/Status
//     PlcTask Inputs/prgEM.fb_KL3403.fbKL3403.byStateCH2 <-> Term 2 (KL3403)/Channel 2/Status
//     PlcTask Inputs/prgEM.fb_KL3403.fbKL3403.byStateCH3 <-> Term 2 (KL3403)/Channel 3/Status
//     PlcTask Inputs/prgEM.fb_KL3403.fbKL3403.iDataInCH1 <-> Term 2 (KL3403)/Channel 1/Daten Ein
//     PlcTask Inputs/prgEM.fb_KL3403.fbKL3403.iDataInCH2 <-> Term 2 (KL3403)/Channel 2/Daten Ein
//     PlcTask Inputs/prgEM.fb_KL3403.fbKL3403.iDataInCH3 <-> Term 2 (KL3403)/Channel 3/Daten Ein
//     PlcTask Inputs/prgEM.iBkStatus <-> Inputs/BoxState
//     PlcTask Outputs/prgEM.fb_KL3403.fbKL3403.byCntrCH1 <-> Term 2 (KL3403)/Channel 1/Kontrolle
//     PlcTask Outputs/prgEM.fb_KL3403.fbKL3403.byCntrCH2 <-> Term 2 (KL3403)/Channel 2/Kontrolle
//     PlcTask Outputs/prgEM.fb_KL3403.fbKL3403.byCntrCH3 <-> Term 2 (KL3403)/Channel 3/Kontrolle

CONFIGURATION SSP_M
    RESOURCE PLC ON TwinCAT3
        TASK FastTask(INTERVAL := T#5ms, PRIORITY := 19);
        TASK PlcTask(INTERVAL := T#10ms, PRIORITY := 20);
        PROGRAM prgPersistent WITH FastTask : prgPersistent;
        PROGRAM prgRWEffIO WITH FastTask : prgRWEffIO;
        PROGRAM prgVarEffIO WITH FastTask : prgVarEffIO;
        PROGRAM prgEM WITH PlcTask : prgEM;
        PROGRAM prgHW WITH PlcTask : prgHW;
        PROGRAM prgEMS WITH PlcTask : prgEMS;
        PROGRAM prgModbus WITH PlcTask : prgModbus;
    END_RESOURCE
END_CONFIGURATION

// ---- FBs/EL3446 FW02 or higher/DUTs/MDP5001_342_O_066CA8C6.TcDUT
TYPE MDP5001_342_O_066CA8C6 :
STRUCT
	MDP5001_342_DPM_Variant_Value_Out_Index_1_REAL	: UINT;
	MDP5001_342_DPM_Variant_Value_Out_Index_2_REAL	: UINT;
	MDP5001_342_DPM_Variant_Value_Out_Index_3_REAL	: UINT;
	MDP5001_342_DPM_Variant_Value_Out_Index_4_ULINT	: UINT;
	MDP5001_342_DPM_Data_Data_1						: UDINT;
	MDP5001_342_DPM_Data_Data_2						: UDINT;
	MDP5001_342_DPM_Data_Data_3						: UDINT;
	MDP5001_342_DPM_Data_Data_4						: UDINT;
	MDP5001_342_DPM_Data_Data_5						: UDINT;
	MDP5001_342_DPM_Data_Data_6						: UDINT;
	MDP5001_342_DPM_Data_Data_7						: UDINT;
	MDP5001_342_DPM_Data_Data_8						: UDINT;
	MDP5001_342_DPM_Data_Data_9						: UDINT;
	MDP5001_342_DPM_Data_Data_10					: UDINT;
	MDP5001_342_DPM_Data_Data_11					: UDINT;
	MDP5001_342_DPM_Data_Data_12					: UDINT;
	MDP5001_342_DPM_Data_Data_13					: UDINT;
	MDP5001_342_DPM_Data_Data_14					: UDINT;
	MDP5001_342_DPM_Data_Data_15					: UDINT;
	MDP5001_342_DPM_Data_Data_16					: UDINT;
	MDP5001_342_DPM_Data_Data_17					: UDINT;
	MDP5001_342_DPM_Data_Data_18					: UDINT;
	MDP5001_342_DPM_Data_Data_19					: UDINT;
	MDP5001_342_DPM_Data_Data_20					: UDINT;
END_STRUCT
END_TYPE

// ---- POUs/prgPersistent.TcPOU
PROGRAM prgPersistent
VAR
	fbUSV		: FB_WritePersistentData_CX81xx;
	
	fb_Reboot		: NT_reboot;
	m_Reboot		: BOOL:=FALSE;
	Int_LiveCount_1min	:INT; 							//{#lynus.ag#()}
	ton_LiveCount	:TON;	
	int_liveCount		:INT;				//{#lynus.ag#()}
END_VAR

fbUSV(
	eSaveModeData:= eUSVSaveMode.eSaveWhenPowerfail, 
	bLoadPersistentDataOk=> , 
	bPowerFailDetect=> , 
	bError=> , 
	bySaveProcess=> , 
	dwStorageLast24h=> , 
	udiErrorCode=> );
	
	
fb_Reboot(	netid := '',
			delay := 2,
			start := m_Reboot);

// 1 min live count
ton_LiveCount(PT:=T#1M);
IF ton_LiveCount.Q THEN
	Int_LiveCount_1min := Int_LiveCount_1min + 1;
	ton_LiveCount.IN := FALSE;
ELSE
	ton_LiveCount.IN := TRUE;
END_IF
// livecount
int_liveCount := int_liveCount+1;

END_PROGRAM

// ---- POUs/prgEM.TcPOU
PROGRAM prgEM
// 06.10.25 Messung am BK9050 ergänzt (EM4) 
VAR
 	fb_EL3443_EM0 		: FB_EM_Beckhoff_EL3443;
	fb_EL3443_EM1 		: FB_EM_Beckhoff_EL3443;		//EL3443 | PDO Assignment "DPM" (DPM: Distributed Power Measurement) |3-phase power measurement terminal with extended functionality
	fb_EL3446_1			: FB_EM_Beckhoff_EL3446;
	fb_EL3446_2			: FB_EM_Beckhoff_EL3446;
  fb_KL3403       : FB_EM_Beckhoff_KL3403;	

  iBkStatus  AT %I* : UINT;
  
	//EM0 (CEE32 3phase Measurement)
	lr_RealPower_EM0		: LREAL;					//{#lynus.ag#()}
	lr_ApparentPower_EM0	: LREAL;					//{#lynus.ag#()}
	lr_ReactivePower_EM0	: LREAL;					//{#lynus.ag#()}
	lr_Frequency_EM0		: LREAL;					//{#lynus.ag#()}
	lr_Voltage_EM0_L1N		: LREAL;					//{#lynus.ag#()}
	lr_Voltage_EM0_L2N		: LREAL;					//{#lynus.ag#()}
	lr_Voltage_EM0_L3N		: LREAL;					//{#lynus.ag#()}
	lr_Voltage_EM0_L1L2		: LREAL;					//{#lynus.ag#()}
	lr_Voltage_EM0_L2L3		: LREAL;					//{#lynus.ag#()}
	lr_Voltage_EM0_L3L1		: LREAL;					//{#lynus.ag#()}
 	lr_Current_EM0_L1		: LREAL;					//{#lynus.ag#()}
	lr_Current_EM0_L2		: LREAL;					//{#lynus.ag#()}
	lr_Current_EM0_L3		: LREAL;					//{#lynus.ag#()}
	
	//EM1 (3phase Measurement, connection Block A)
	lr_RealPower_EM1		: LREAL;					//{#lynus.ag#()}
	lr_ApparentPower_EM1	: LREAL;					//{#lynus.ag#()}
	lr_ReactivePower_EM1	: LREAL;					//{#lynus.ag#()}
	lr_Frequency_EM1		: LREAL;					//{#lynus.ag#()}
	lr_Voltage_EM1_L1N		: LREAL;					//{#lynus.ag#()}
	lr_Voltage_EM1_L2N		: LREAL;					//{#lynus.ag#()}
	lr_Voltage_EM1_L3N		: LREAL;					//{#lynus.ag#()}
	lr_Voltage_EM1_L1L2		: LREAL;					//{#lynus.ag#()}
	lr_Voltage_EM1_L2L3		: LREAL;					//{#lynus.ag#()}
	lr_Voltage_EM1_L3L1		: LREAL;					//{#lynus.ag#()}
 	lr_Current_EM1_L1		: LREAL;					//{#lynus.ag#()}
	lr_Current_EM1_L2		: LREAL;					//{#lynus.ag#()}
	lr_Current_EM1_L3		: LREAL;					//{#lynus.ag#()}
	
	//EM2, connection Blocks B-C
	lrPower_EM2_1		: LREAL;						//{#lynus.ag#()}
	lrPower_EM2_2		: LREAL;						//{#lynus.ag#()}
	lrPower_EM2_3		: LREAL;						//{#lynus.ag#()}
	lrPower_EM2_4		: LREAL;						//{#lynus.ag#()}
	lrPower_EM2_5		: LREAL;						//{#lynus.ag#()}
	lrPower_EM2_6		: LREAL;						//{#lynus.ag#()}
	lrPower_EM2_3p1		: LREAL;						//{#lynus.ag#()}
	lrPower_EM2_3p2		: LREAL;						//{#lynus.ag#()}
	
	//EM3, connection Blocks D-E
	lrPower_EM3_1		: LREAL;						//{#lynus.ag#()}
	lrPower_EM3_2		: LREAL;						//{#lynus.ag#()}
	lrPower_EM3_3		: LREAL;						//{#lynus.ag#()}
	lrPower_EM3_4		: LREAL;						//{#lynus.ag#()}
	lrPower_EM3_5		: LREAL;						//{#lynus.ag#()}
	lrPower_EM3_6		: LREAL;						//{#lynus.ag#()}
	lrPower_EM3_3p1		: LREAL;						//{#lynus.ag#()}
	lrPower_EM3_3p2		: LREAL;						//{#lynus.ag#()}

	//EM3, connection BK9050
	lrPower_EM4_1		: LREAL;						//{#lynus.ag#()}
	lrPower_EM4_2		: LREAL;						//{#lynus.ag#()}
	lrPower_EM4_3		: LREAL;						//{#lynus.ag#()}
	lrPower_EM4_3p1		: LREAL;						//{#lynus.ag#()}
END_VAR

VAR_INPUT
	stEL3443_IO_1 						: MDP5001_341_7CD731EE;
	stEL3443_IO_2 						: MDP5001_341_7CD731EE;
	stEL3446_IO_1 						: MDP5001_342_066CA8C6; 
	stEL3446_IO_2 						: MDP5001_342_066CA8C6;	
END_VAR

VAR PERSISTENT
	uiCurrentTransformerRatio_EM0	:UINT:=32;
	uiCurrentTransformerRatio_EM1	:UINT:=300;				//{#lynus.ag#()}
	lr_EnergyCounter_EM0	: LREAL;
	lr_EnergyCounter_EM1	: LREAL;
	
	ui_PhaseSelector_EM1_1 : UINT := 1;						//{#lynus.ag#()}
	ui_PhaseSelector_EM1_2 : UINT := 2;						//{#lynus.ag#()}
	ui_PhaseSelector_EM1_3 : UINT := 3;						//{#lynus.ag#()}
	ui_PhaseSelector_EM2_1 : UINT := 1;						//{#lynus.ag#()}
	ui_PhaseSelector_EM2_2 : UINT := 2;						//{#lynus.ag#()}
	ui_PhaseSelector_EM2_3 : UINT := 3;						//{#lynus.ag#()}
	ui_PhaseSelector_EM2_4 : UINT := 1;						//{#lynus.ag#()}
	ui_PhaseSelector_EM2_5 : UINT := 2;						//{#lynus.ag#()}
	ui_PhaseSelector_EM2_6 : UINT := 3;						//{#lynus.ag#()}
	ui_PhaseSelector_EM3_1 : UINT := 1;						//{#lynus.ag#()}
	ui_PhaseSelector_EM3_2 : UINT := 2;						//{#lynus.ag#()}
	ui_PhaseSelector_EM3_3 : UINT := 3;						//{#lynus.ag#()}
	ui_PhaseSelector_EM3_4 : UINT := 1;						//{#lynus.ag#()}
	ui_PhaseSelector_EM3_5 : UINT := 2;						//{#lynus.ag#()}
	ui_PhaseSelector_EM3_6 : UINT := 3;						//{#lynus.ag#()}
	
	uiCurrentTransformerRatio_EM1_1	: UINT := 300;				//{#lynus.ag#()}
	uiCurrentTransformerRatio_EM1_2	: UINT := 300;				//{#lynus.ag#()}
	uiCurrentTransformerRatio_EM1_3	: UINT := 300;				//{#lynus.ag#()}
	uiCurrentTransformerRatio_EM2_1	: UINT := 300;				//{#lynus.ag#()}
	uiCurrentTransformerRatio_EM2_2	: UINT := 300;				//{#lynus.ag#()}
	uiCurrentTransformerRatio_EM2_3	: UINT := 300;				//{#lynus.ag#()}
	uiCurrentTransformerRatio_EM2_4	: UINT := 300;				//{#lynus.ag#()}
	uiCurrentTransformerRatio_EM2_5	: UINT := 300;				//{#lynus.ag#()}
	uiCurrentTransformerRatio_EM2_6	: UINT := 300;				//{#lynus.ag#()}
	uiCurrentTransformerRatio_EM3_1	: UINT := 300;				//{#lynus.ag#()}
	uiCurrentTransformerRatio_EM3_2	: UINT := 300;				//{#lynus.ag#()}
	uiCurrentTransformerRatio_EM3_3	: UINT := 300;				//{#lynus.ag#()}
	uiCurrentTransformerRatio_EM3_4	: UINT := 300;				//{#lynus.ag#()}
	uiCurrentTransformerRatio_EM3_5	: UINT := 300;				//{#lynus.ag#()}
	uiCurrentTransformerRatio_EM3_6	: UINT := 300;				//{#lynus.ag#()}
	uiCurrentTransformerRatio_EM4_1	: UINT := 300;				//{#lynus.ag#()}
	uiCurrentTransformerRatio_EM4_2	: UINT := 300;				//{#lynus.ag#()}
	uiCurrentTransformerRatio_EM4_3	: UINT := 300;				//{#lynus.ag#()}
	
	b_Invers_EM1_1	:	BOOL := FALSE;							//{#lynus.ag#()}
	b_Invers_EM1_2	:	BOOL := FALSE;							//{#lynus.ag#()}
	b_Invers_EM1_3	:	BOOL := FALSE;							//{#lynus.ag#()}
	b_Invers_EM2_1	:	BOOL := FALSE;							//{#lynus.ag#()}
	b_Invers_EM2_2	:	BOOL := FALSE;							//{#lynus.ag#()}
	b_Invers_EM2_3	:	BOOL := FALSE;							//{#lynus.ag#()}
	b_Invers_EM2_4	:	BOOL := FALSE;							//{#lynus.ag#()}
	b_Invers_EM2_5	:	BOOL := FALSE;							//{#lynus.ag#()}
	b_Invers_EM2_6	:	BOOL := FALSE;							//{#lynus.ag#()}
	b_Invers_EM3_1	:	BOOL := FALSE;							//{#lynus.ag#()}
	b_Invers_EM3_2	:	BOOL := FALSE;							//{#lynus.ag#()}
	b_Invers_EM3_3	:	BOOL := FALSE;							//{#lynus.ag#()}
	b_Invers_EM3_4	:	BOOL := FALSE;							//{#lynus.ag#()}
	b_Invers_EM3_5	:	BOOL := FALSE;							//{#lynus.ag#()}
	b_Invers_EM3_6	:	BOOL := FALSE;							//{#lynus.ag#()}
	b_Invers_EM4_1	:	BOOL := FALSE;							//{#lynus.ag#()}
	b_Invers_EM4_2	:	BOOL := FALSE;							//{#lynus.ag#()}
	b_Invers_EM4_3	:	BOOL := FALSE;							//{#lynus.ag#()}

END_VAR

//EM0 (CEE32 3phase Measurement)
fb_EL3443_EM0(
	bEnable 	:= TRUE, 
	bInvers_CH1 := , 
	bInvers_CH2	:= , 
	bInvers_CH3	:= , 
	uiCurrentTransformerRatio:= uiCurrentTransformerRatio_EM0, 
	nSlaveAddr 	:= 1001,
	stEL3443_IO := ,
	pDpmData=> , 
	stDataEMPower=> , 
	stDataEMCounter=> , 
	stDataEMPowerRealTime=> , 
	stDataEMCounterRealTime=> );

fb_EL3443_EM0.stEL3443_IO.MDP5001_341_Input := stEL3443_IO_1.MDP5001_341_Input;
stEL3443_IO_1.MDP5001_341_Output	:= fb_EL3443_EM0.stEL3443_IO.MDP5001_341_Output;
 	
lr_RealPower_EM0 			:= fb_EL3443_EM0.stDataEMPower.lrPowerTotal; 	
lr_ApparentPower_EM0 		:= fb_EL3443_EM0.stDataEMPower.lrApparentPowerTotal;
lr_ReactivePower_EM0		:= fb_EL3443_EM0.stDataEMPower.lrReactivePowerTotal;
lr_Frequency_EM0			:= fb_EL3443_EM0.stDataEMPower.lrFrequency;
lr_Voltage_EM0_L1N			:= fb_EL3443_EM0.stDataEMPower.lrVoltageL1N;
lr_Voltage_EM0_L2N			:= fb_EL3443_EM0.stDataEMPower.lrVoltageL2N;
lr_Voltage_EM0_L3N			:= fb_EL3443_EM0.stDataEMPower.lrVoltageL3N;
lr_Voltage_EM0_L1L2			:= fb_EL3443_EM0.stDataEMPower.lrVoltageL1L2;
lr_Voltage_EM0_L2L3			:= fb_EL3443_EM0.stDataEMPower.lrVoltageL2L3;
lr_Voltage_EM0_L3L1			:= fb_EL3443_EM0.stDataEMPower.lrVoltageL3L1;
lr_EnergyCounter_EM0		:= fb_EL3443_EM0.stDataEMCounter.lrTotalCounterEnergy_Consumption;
lr_Current_EM0_L1			:= fb_EL3443_EM0.stDataEMPower.lrCurrentL1;
lr_Current_EM0_L2			:= fb_EL3443_EM0.stDataEMPower.lrCurrentL2;
lr_Current_EM0_L3			:= fb_EL3443_EM0.stDataEMPower.lrCurrentL3;


//EM1 (for 3-phase Measurement, connection Block A)
fb_EL3443_EM1(
	bEnable 	:= TRUE, 
	bInvers_CH1 := b_Invers_EM1_1, 
	bInvers_CH2	:= b_Invers_EM1_2, 
	bInvers_CH3	:= b_Invers_EM1_3, 
	uiCurrentTransformerRatio:= uiCurrentTransformerRatio_EM1,
	nSlaveAddr 	:= 1002,
	stEL3443_IO := ,
	pDpmData=> , 
	stDataEMPower=> , 
	stDataEMCounter=> , 
	stDataEMPowerRealTime=> , 
	stDataEMCounterRealTime=> );

fb_EL3443_EM1.stEL3443_IO.MDP5001_341_Input := stEL3443_IO_2.MDP5001_341_Input;
stEL3443_IO_2.MDP5001_341_Output	:= fb_EL3443_EM1.stEL3443_IO.MDP5001_341_Output;
 	
lr_RealPower_EM1 			:= fb_EL3443_EM1.stDataEMPower.lrPowerTotal; 	
lr_ApparentPower_EM1 		:= fb_EL3443_EM1.stDataEMPower.lrApparentPowerTotal;
lr_ReactivePower_EM1		:= fb_EL3443_EM1.stDataEMPower.lrReactivePowerTotal;
lr_Frequency_EM1			:= fb_EL3443_EM1.stDataEMPower.lrFrequency;
lr_Voltage_EM1_L1N			:= fb_EL3443_EM1.stDataEMPower.lrVoltageL1N;
lr_Voltage_EM1_L2N			:= fb_EL3443_EM1.stDataEMPower.lrVoltageL2N;
lr_Voltage_EM1_L3N			:= fb_EL3443_EM1.stDataEMPower.lrVoltageL3N;
lr_Voltage_EM1_L1L2			:= fb_EL3443_EM1.stDataEMPower.lrVoltageL1L2;
lr_Voltage_EM1_L2L3			:= fb_EL3443_EM1.stDataEMPower.lrVoltageL2L3;
lr_Voltage_EM1_L3L1			:= fb_EL3443_EM1.stDataEMPower.lrVoltageL3L1;
lr_EnergyCounter_EM1		:= fb_EL3443_EM1.stDataEMCounter.lrTotalCounterEnergy_Consumption;
lr_Current_EM1_L1			:= fb_EL3443_EM1.stDataEMPower.lrCurrentL1;
lr_Current_EM1_L2			:= fb_EL3443_EM1.stDataEMPower.lrCurrentL2;
lr_Current_EM1_L3			:= fb_EL3443_EM1.stDataEMPower.lrCurrentL3;

//EM2 (for single Phase Measurements, connection Block B-C)
fb_EL3446_1(
	bEnable:= TRUE , 
	bEnableVariantValues:= TRUE, 
	pDpmData:= fb_EL3443_EM1.pDpmData, 
	nSlaveAddr:= 1003, 
	bInvers_CH1:= b_Invers_EM2_1, 
	bInvers_CH2:= b_Invers_EM2_2, 
	bInvers_CH3:= b_Invers_EM2_3, 
	bInvers_CH4:= b_Invers_EM2_4, 
	bInvers_CH5:= b_Invers_EM2_5, 
	bInvers_CH6:= b_Invers_EM2_6, 
	uiCurrentTransformerRatio_CH1:= uiCurrentTransformerRatio_EM2_1, 
	uiCurrentTransformerRatio_CH2:= uiCurrentTransformerRatio_EM2_2, 
	uiCurrentTransformerRatio_CH3:= uiCurrentTransformerRatio_EM2_3, 
	uiCurrentTransformerRatio_CH4:= uiCurrentTransformerRatio_EM2_4, 
	uiCurrentTransformerRatio_CH5:= uiCurrentTransformerRatio_EM2_5, 
	uiCurrentTransformerRatio_CH6:= uiCurrentTransformerRatio_EM2_6, 
	uiVoltagePhaseSelector_CH1:= ui_PhaseSelector_EM2_1, 
	uiVoltagePhaseSelector_CH2:= ui_PhaseSelector_EM2_2, 
	uiVoltagePhaseSelector_CH3:= ui_PhaseSelector_EM2_3, 
	uiVoltagePhaseSelector_CH4:= ui_PhaseSelector_EM2_4, 
	uiVoltagePhaseSelector_CH5:= ui_PhaseSelector_EM2_5, 
	uiVoltagePhaseSelector_CH6:= ui_PhaseSelector_EM2_6, 
	bEnable3PhaseCH13:= FALSE, 
	bEnable3PhaseCH46:= FALSE, 
	stDataEMPowerRealTime:= fb_EL3443_EM1.stDataEMPowerRealTime, 
	stEL3446_IO := ,
	stDataEMPower_CH1=> , 
	stDataEMCounter_CH1=> , 
	stDataEMPowerRealTime_CH1=> , 
	stDataEMCounterRealTime_CH1=> , 
	stDataEMPower_CH2=> , 
	stDataEMCounter_CH2=> , 
	stDataEMPowerRealTime_CH2=> , 
	stDataEMCounterRealTime_CH2=> , 
	stDataEMPower_CH3=> , 
	stDataEMCounter_CH3=> , 
	stDataEMPowerRealTime_CH3=> , 
	stDataEMCounterRealTime_CH3=> , 
	stDataEMPower_CH4=> , 
	stDataEMCounter_CH4=> , 
	stDataEMPowerRealTime_CH4=> , 
	stDataEMCounterRealTime_CH4=> , 
	stDataEMPower_CH5=> , 
	stDataEMCounter_CH5=> , 
	stDataEMPowerRealTime_CH5=> , 
	stDataEMCounterRealTime_CH5=> , 
	stDataEMPower_CH6=> , 
	stDataEMCounter_CH6=> , 
	stDataEMPowerRealTime_CH6=> , 
	stDataEMCounterRealTime_CH6=> );
fb_EL3446_1.stEL3446_IO.MDP5001_342_Input := stEL3446_IO_1.MDP5001_342_Input;
stEL3446_IO_1.MDP5001_342_Output := 	fb_EL3446_1.stEL3446_IO.MDP5001_342_Output;

lrPower_EM2_1				:= 	LIMIT(0,fb_EL3446_1.stDataEMPower_CH1.lrPowerTotal,1000);
lrPower_EM2_2				:= 	LIMIT(0,fb_EL3446_1.stDataEMPower_CH2.lrPowerTotal,1000);
lrPower_EM2_3				:= 	LIMIT(0,fb_EL3446_1.stDataEMPower_CH3.lrPowerTotal,1000);
lrPower_EM2_4				:= 	LIMIT(0,fb_EL3446_1.stDataEMPower_CH4.lrPowerTotal,1000);
lrPower_EM2_5				:= 	LIMIT(0,fb_EL3446_1.stDataEMPower_CH5.lrPowerTotal,1000);
lrPower_EM2_6				:= 	LIMIT(0,fb_EL3446_1.stDataEMPower_CH6.lrPowerTotal,1000);

lrPower_EM2_3p1 			:= lrPower_EM2_1 + lrPower_EM2_2 + lrPower_EM2_3;
lrPower_EM2_3p2 			:= lrPower_EM2_4 + lrPower_EM2_5 + lrPower_EM2_6;

(*
lr_EnergyCounter_EM1	:= 	fb_EL3446_1.stDataEMCounter_CH1.lrTotalCounterEnergy_Consumption;
lr_EnergyCounter_EM2	:= 	fb_EL3446_1.stDataEMCounter_CH2.lrTotalCounterEnergy_Consumption;
lr_EnergyCounter_EM3	:= 	fb_EL3446_1.stDataEMCounter_CH3.lrTotalCounterEnergy_Consumption;
lr_EnergyCounter_EM4	:= 	fb_EL3446_1.stDataEMCounter_CH4.lrTotalCounterEnergy_Consumption;
lr_EnergyCounter_EM5	:= 	fb_EL3446_1.stDataEMCounter_CH5.lrTotalCounterEnergy_Consumption;
lr_EnergyCounter_EM6	:= 	fb_EL3446_1.stDataEMCounter_CH6.lrTotalCounterEnergy_Consumption;
*)

//EM3 (for single Phase Measurements, connection Block D-E)
fb_EL3446_2(
	bEnable:= TRUE , 
	bEnableVariantValues:= TRUE, 
	pDpmData:= fb_EL3443_EM1.pDpmData, 
	nSlaveAddr:= 1004, 
	bInvers_CH1:= b_Invers_EM3_1, 
	bInvers_CH2:= b_Invers_EM3_2, 
	bInvers_CH3:= b_Invers_EM3_3, 
	bInvers_CH4:= b_Invers_EM3_4, 
	bInvers_CH5:= b_Invers_EM3_5, 
	bInvers_CH6:= b_Invers_EM3_6, 
	uiCurrentTransformerRatio_CH1:= uiCurrentTransformerRatio_EM3_1, 
	uiCurrentTransformerRatio_CH2:= uiCurrentTransformerRatio_EM3_2, 
	uiCurrentTransformerRatio_CH3:= uiCurrentTransformerRatio_EM3_3, 
	uiCurrentTransformerRatio_CH4:= uiCurrentTransformerRatio_EM3_4, 
	uiCurrentTransformerRatio_CH5:= uiCurrentTransformerRatio_EM3_5, 
	uiCurrentTransformerRatio_CH6:= uiCurrentTransformerRatio_EM3_6, 
	uiVoltagePhaseSelector_CH1:= ui_PhaseSelector_EM3_1, 
	uiVoltagePhaseSelector_CH2:= ui_PhaseSelector_EM3_2, 
	uiVoltagePhaseSelector_CH3:= ui_PhaseSelector_EM3_3, 
	uiVoltagePhaseSelector_CH4:= ui_PhaseSelector_EM3_4, 
	uiVoltagePhaseSelector_CH5:= ui_PhaseSelector_EM3_5, 
	uiVoltagePhaseSelector_CH6:= ui_PhaseSelector_EM3_6, 
	bEnable3PhaseCH13:= FALSE, 
	bEnable3PhaseCH46:= FALSE, 
	stDataEMPowerRealTime:= fb_EL3443_EM1.stDataEMPowerRealTime, 
	stEL3446_IO := ,
	stDataEMPower_CH1=> , 
	stDataEMCounter_CH1=> , 
	stDataEMPowerRealTime_CH1=> , 
	stDataEMCounterRealTime_CH1=> , 
	stDataEMPower_CH2=> , 
	stDataEMCounter_CH2=> , 
	stDataEMPowerRealTime_CH2=> , 
	stDataEMCounterRealTime_CH2=> , 
	stDataEMPower_CH3=> , 
	stDataEMCounter_CH3=> , 
	stDataEMPowerRealTime_CH3=> , 
	stDataEMCounterRealTime_CH3=> , 
	stDataEMPower_CH4=> , 
	stDataEMCounter_CH4=> , 
	stDataEMPowerRealTime_CH4=> , 
	stDataEMCounterRealTime_CH4=> , 
	stDataEMPower_CH5=> , 
	stDataEMCounter_CH5=> , 
	stDataEMPowerRealTime_CH5=> , 
	stDataEMCounterRealTime_CH5=> , 
	stDataEMPower_CH6=> , 
	stDataEMCounter_CH6=> , 
	stDataEMPowerRealTime_CH6=> , 
	stDataEMCounterRealTime_CH6=> );
fb_EL3446_2.stEL3446_IO.MDP5001_342_Input := stEL3446_IO_2.MDP5001_342_Input;
stEL3446_IO_2.MDP5001_342_Output := 	fb_EL3446_2.stEL3446_IO.MDP5001_342_Output;

lrPower_EM3_1				:= 	LIMIT(0,fb_EL3446_2.stDataEMPower_CH1.lrPowerTotal,1000);
lrPower_EM3_2				:= 	LIMIT(0,fb_EL3446_2.stDataEMPower_CH2.lrPowerTotal,1000);
lrPower_EM3_3				:= 	LIMIT(0,fb_EL3446_2.stDataEMPower_CH3.lrPowerTotal,1000);
lrPower_EM3_4				:= 	LIMIT(0,fb_EL3446_2.stDataEMPower_CH4.lrPowerTotal,1000);
lrPower_EM3_5				:= 	LIMIT(0,fb_EL3446_2.stDataEMPower_CH5.lrPowerTotal,1000);
lrPower_EM3_6				:= 	LIMIT(0,fb_EL3446_2.stDataEMPower_CH6.lrPowerTotal,1000);

lrPower_EM3_3p1 			:= lrPower_EM3_1 + lrPower_EM3_2 + lrPower_EM3_3;
lrPower_EM3_3p2 			:= lrPower_EM3_4 + lrPower_EM3_5 + lrPower_EM3_6;

//EM4 (for single Phase Measurements, connection BK9050)
fb_KL3403(
	bEnable:= TRUE, 
	bChannel1Invers:= b_Invers_EM4_1, 
	bChannel2Invers:= b_Invers_EM4_2, 
	bChannel3Invers:= b_Invers_EM4_3, 
	uiCurrentTransformerRatioL1:= uiCurrentTransformerRatio_EM4_1, 
	uiCurrentTransformerRatioL2:= uiCurrentTransformerRatio_EM4_2, 
	uiCurrentTransformerRatioL3:= uiCurrentTransformerRatio_EM4_3, 
	uiKBusState_IN:= iBkStatus, 
	stDataEMPower=> , 
	stDataEMCounter=> , 
	stDataEMPowerRealTime=> , 
	stDataEMCounterRealTime=> , 
	diNrOfEM_OUT=> );

lrPower_EM4_1				:= 	LIMIT(0,fb_KL3403.stDataEMPower.lrPowerL1,1000);
lrPower_EM4_2				:= 	LIMIT(0,fb_KL3403.stDataEMPower.lrPowerL2,1000);
lrPower_EM4_3				:= 	LIMIT(0,fb_KL3403.stDataEMPower.lrPowerL3,1000);

lrPower_EM3_3p1 		:= lrPower_EM4_1 + lrPower_EM4_2 + lrPower_EM4_3;

END_PROGRAM

// ---- POUs/prgHW.TcPOU
PROGRAM prgHW
VAR

	// IOs for EL3443
	{attribute 'TcLinkTo' := 'TIID^Device 2 (EtherCAT)^Term 1 (EK1200)^Term 6 (EL3443)^L1 Status^Voltage Sign Bit'}
	MDP5001_341_L1_Status_Voltage_Sign_Bit   	AT%I*  : BOOL;  // linked via attribute 
	{attribute 'TcLinkTo' := 'TIID^Device 2 (EtherCAT)^Term 1 (EK1200)^Term 6 (EL3443)^L1 Status^Overvoltage'}
	MDP5001_341_L1_Status_Overvoltage			AT%I*  : BOOL;  // linked via attribute 
	{attribute 'TcLinkTo' := 'TIID^Device 2 (EtherCAT)^Term 1 (EK1200)^Term 6 (EL3443)^L1 Status^Overcurrent'}
	MDP5001_341_L1_Status_Overcurrent			AT%I*  : BOOL;  // linked via attribute 
	{attribute 'TcLinkTo' := 'TIID^Device 2 (EtherCAT)^Term 1 (EK1200)^Term 6 (EL3443)^L1 Status^Inaccurate Voltage'}	
	MDP5001_341_L1_Status_Inaccurate_Voltage	AT%I*  : BOOL;  // linked via attribute 
	{attribute 'TcLinkTo' := 'TIID^Device 2 (EtherCAT)^Term 1 (EK1200)^Term 6 (EL3443)^L1 Status^Inaccurate Current'}
	MDP5001_341_L1_Status_Inaccurate_Current	AT%I*  : BOOL;  // linked via attribute 	
	{attribute 'TcLinkTo' := 'TIID^Device 2 (EtherCAT)^Term 1 (EK1200)^Term 6 (EL3443)^L1 Status^Voltage Guard Warning'}
	MDP5001_341_L1_Status_Voltage_Guard_Warning	AT%I*  : BOOL;  // linked via attribute
	{attribute 'TcLinkTo' := 'TIID^Device 2 (EtherCAT)^Term 1 (EK1200)^Term 6 (EL3443)^L1 Status^Voltage Guard Error'}
	MDP5001_341_L1_Status_Voltage_Guard_Error	AT%I*  : BOOL;  // linked via attribute
	{attribute 'TcLinkTo' := 'TIID^Device 2 (EtherCAT)^Term 1 (EK1200)^Term 6 (EL3443)^L1 Status^Current Guard Warning'}
	MDP5001_341_L1_Status_Current_Guard_Warning AT%I*  : BOOL;  // linked via attribute
	{attribute 'TcLinkTo' := 'TIID^Device 2 (EtherCAT)^Term 1 (EK1200)^Term 6 (EL3443)^L1 Status^Current Guard Error'}
	MDP5001_341_L1_Status_Current_Guard_Error	AT%I*  : BOOL;  // linked via attribute
	{attribute 'TcLinkTo' := 'TIID^Device 2 (EtherCAT)^Term 1 (EK1200)^Term 6 (EL3443)^L1 Status^TxPDO Toggle'}
	MDP5001_341_L1_Status_TxPDO_Toggle			AT%I*  : BOOL;  // linked via attribute
	{attribute 'TcLinkTo' := 'TIID^Device 2 (EtherCAT)^Term 1 (EK1200)^Term 6 (EL3443)^L1 Basic^Voltage'}
	MDP5001_341_L1_Basic_Voltage				AT%I*  : REAL;		// linked via attribute 
	{attribute 'TcLinkTo' := 'TIID^Device 2 (EtherCAT)^Term 1 (EK1200)^Term 6 (EL3443)^L1 Basic^Current'}
	MDP5001_341_L1_Basic_Current				AT%I*  : REAL;		// linked via attribute 
	{attribute 'TcLinkTo' := 'TIID^Device 2 (EtherCAT)^Term 1 (EK1200)^Term 6 (EL3443)^L1 Power^Active Power'}
	MDP5001_341_L1_Power_Active_Power			AT%I*  : REAL;		// linked via attribute 
	{attribute 'TcLinkTo' := 'TIID^Device 2 (EtherCAT)^Term 1 (EK1200)^Term 6 (EL3443)^L1 Power^Apparent Power'}
	MDP5001_341_L1_Power_Apparent_Power			AT%I* : REAL;		// linked via attribute 
	{attribute 'TcLinkTo' := 'TIID^Device 2 (EtherCAT)^Term 1 (EK1200)^Term 6 (EL3443)^L1 Power^Reactive Power'}
	MDP5001_341_L1_Power_Reactive_Power			AT%I* : REAL;		// linked via attribute 
	{attribute 'TcLinkTo' := 'TIID^Device 2 (EtherCAT)^Term 1 (EK1200)^Term 6 (EL3443)^L1 Power^Power Factor'}
	MDP5001_341_L1_Power_Power_Factor			AT%I* : REAL;		// linked via attribute 
	{attribute 'TcLinkTo' := 'TIID^Device 2 (EtherCAT)^Term 1 (EK1200)^Term 6 (EL3443)^L2 Status^Voltage Sign Bit'}
	MDP5001_341_L2_Status_Voltage_Sign_Bit   	AT%I*  : BOOL;  // linked via attribute 
	{attribute 'TcLinkTo' := 'TIID^Device 2 (EtherCAT)^Term 1 (EK1200)^Term 6 (EL3443)^L2 Status^Overvoltage'}
	MDP5001_341_L2_Status_Overvoltage			AT%I*  : BOOL;  // linked via attribute 
	{attribute 'TcLinkTo' := 'TIID^Device 2 (EtherCAT)^Term 1 (EK1200)^Term 6 (EL3443)^L2 Status^Overcurrent'}
	MDP5001_341_L2_Status_Overcurrent			AT%I*  : BOOL;  // linked via attribute 
	{attribute 'TcLinkTo' := 'TIID^Device 2 (EtherCAT)^Term 1 (EK1200)^Term 6 (EL3443)^L2 Status^Inaccurate Voltage'}	
	MDP5001_341_L2_Status_Inaccurate_Voltage	AT%I*  : BOOL;  // linked via attribute 
	{attribute 'TcLinkTo' := 'TIID^Device 2 (EtherCAT)^Term 1 (EK1200)^Term 6 (EL3443)^L2 Status^Inaccurate Current'}
	MDP5001_341_L2_Status_Inaccurate_Current	AT%I*  : BOOL;  // linked via attribute 	
	{attribute 'TcLinkTo' := 'TIID^Device 2 (EtherCAT)^Term 1 (EK1200)^Term 6 (EL3443)^L2 Status^Voltage Guard Warning'}
	MDP5001_341_L2_Status_Voltage_Guard_Warning	AT%I*  : BOOL;  // linked via attribute
	{attribute 'TcLinkTo' := 'TIID^Device 2 (EtherCAT)^Term 1 (EK1200)^Term 6 (EL3443)^L2 Status^Voltage Guard Error'}
	MDP5001_341_L2_Status_Voltage_Guard_Error	AT%I*  : BOOL;  // linked via attribute
	{attribute 'TcLinkTo' := 'TIID^Device 2 (EtherCAT)^Term 1 (EK1200)^Term 6 (EL3443)^L2 Status^Current Guard Warning'}
	MDP5001_341_L2_Status_Current_Guard_Warning AT%I*  : BOOL;  // linked via attribute
	{attribute 'TcLinkTo' := 'TIID^Device 2 (EtherCAT)^Term 1 (EK1200)^Term 6 (EL3443)^L2 Status^Current Guard Error'}
	MDP5001_341_L2_Status_Current_Guard_Error	AT%I*  : BOOL;  // linked via attribute
	{attribute 'TcLinkTo' := 'TIID^Device 2 (EtherCAT)^Term 1 (EK1200)^Term 6 (EL3443)^L2 Status^TxPDO Toggle'}
	MDP5001_341_L2_Status_TxPDO_Toggle			AT%I*  : BOOL;  // linked via attribute
	{attribute 'TcLinkTo' := 'TIID^Device 2 (EtherCAT)^Term 1 (EK1200)^Term 6 (EL3443)^L2 Basic^Voltage'}
	MDP5001_341_L2_Basic_Voltage				AT%I* : REAL;		// linked via attribute 
	{attribute 'TcLinkTo' := 'TIID^Device 2 (EtherCAT)^Term 1 (EK1200)^Term 6 (EL3443)^L2 Basic^Current'}
	MDP5001_341_L2_Basic_Current				AT%I* : REAL;		// linked via attribute 
	{attribute 'TcLinkTo' := 'TIID^Device 2 (EtherCAT)^Term 1 (EK1200)^Term 6 (EL3443)^L2 Power^Active Power'}
	MDP5001_341_L2_Power_Active_Power			AT%I* : REAL;		// linked via attribute 
	{attribute 'TcLinkTo' := 'TIID^Device 2 (EtherCAT)^Term 1 (EK1200)^Term 6 (EL3443)^L2 Power^Apparent Power'}
	MDP5001_341_L2_Power_Apparent_Power			AT%I* : REAL;		// linked via attribute 
	{attribute 'TcLinkTo' := 'TIID^Device 2 (EtherCAT)^Term 1 (EK1200)^Term 6 (EL3443)^L2 Power^Reactive Power'}
	MDP5001_341_L2_Power_Reactive_Power			AT%I* : REAL;		// linked via attribute 
	{attribute 'TcLinkTo' := 'TIID^Device 2 (EtherCAT)^Term 1 (EK1200)^Term 6 (EL3443)^L2 Power^Power Factor'}
	MDP5001_341_L2_Power_Power_Factor			AT%I* : REAL;		// linked via attribute 
	{attribute 'TcLinkTo' := 'TIID^Device 2 (EtherCAT)^Term 1 (EK1200)^Term 6 (EL3443)^L3 Status^Voltage Sign Bit'}
	MDP5001_341_L3_Status_Voltage_Sign_Bit   	AT%I*  : BOOL;  // linked via attribute 
	{attribute 'TcLinkTo' := 'TIID^Device 2 (EtherCAT)^Term 1 (EK1200)^Term 6 (EL3443)^L3 Status^Overvoltage'}
	MDP5001_341_L3_Status_Overvoltage			AT%I*  : BOOL;  // linked via attribute 
	{attribute 'TcLinkTo' := 'TIID^Device 2 (EtherCAT)^Term 1 (EK1200)^Term 6 (EL3443)^L3 Status^Overcurrent'}
	MDP5001_341_L3_Status_Overcurrent			AT%I*  : BOOL;  // linked via attribute 
	{attribute 'TcLinkTo' := 'TIID^Device 2 (EtherCAT)^Term 1 (EK1200)^Term 6 (EL3443)^L3 Status^Inaccurate Voltage'}	
	MDP5001_341_L3_Status_Inaccurate_Voltage	AT%I*  : BOOL;  // linked via attribute 
	{attribute 'TcLinkTo' := 'TIID^Device 2 (EtherCAT)^Term 1 (EK1200)^Term 6 (EL3443)^L3 Status^Inaccurate Current'}
	MDP5001_341_L3_Status_Inaccurate_Current	AT%I*  : BOOL;  // linked via attribute 	
	{attribute 'TcLinkTo' := 'TIID^Device 2 (EtherCAT)^Term 1 (EK1200)^Term 6 (EL3443)^L3 Status^Voltage Guard Warning'}
	MDP5001_341_L3_Status_Voltage_Guard_Warning	AT%I*  : BOOL;  // linked via attribute
	{attribute 'TcLinkTo' := 'TIID^Device 2 (EtherCAT)^Term 1 (EK1200)^Term 6 (EL3443)^L3 Status^Voltage Guard Error'}
	MDP5001_341_L3_Status_Voltage_Guard_Error	AT%I*  : BOOL;  // linked via attribute
	{attribute 'TcLinkTo' := 'TIID^Device 2 (EtherCAT)^Term 1 (EK1200)^Term 6 (EL3443)^L3 Status^Current Guard Warning'}
	MDP5001_341_L3_Status_Current_Guard_Warning AT%I*  : BOOL;  // linked via attribute
	{attribute 'TcLinkTo' := 'TIID^Device 2 (EtherCAT)^Term 1 (EK1200)^Term 6 (EL3443)^L3 Status^Current Guard Error'}
	MDP5001_341_L3_Status_Current_Guard_Error	AT%I*  : BOOL;  // linked via attribute
	{attribute 'TcLinkTo' := 'TIID^Device 2 (EtherCAT)^Term 1 (EK1200)^Term 6 (EL3443)^L3 Status^TxPDO Toggle'}
	MDP5001_341_L3_Status_TxPDO_Toggle			AT%I*  : BOOL;  // linked via attribute
	{attribute 'TcLinkTo' := 'TIID^Device 2 (EtherCAT)^Term 1 (EK1200)^Term 6 (EL3443)^L3 Basic^Voltage'}
	MDP5001_341_L3_Basic_Voltage				AT%I* : REAL;		// linked via attribute 
	{attribute 'TcLinkTo' := 'TIID^Device 2 (EtherCAT)^Term 1 (EK1200)^Term 6 (EL3443)^L3 Basic^Current'}
	MDP5001_341_L3_Basic_Current				AT%I* : REAL;		// linked via attribute 
	{attribute 'TcLinkTo' := 'TIID^Device 2 (EtherCAT)^Term 1 (EK1200)^Term 6 (EL3443)^L3 Power^Active Power'}
	MDP5001_341_L3_Power_Active_Power			AT%I* : REAL;		// linked via attribute 
	{attribute 'TcLinkTo' := 'TIID^Device 2 (EtherCAT)^Term 1 (EK1200)^Term 6 (EL3443)^L3 Power^Apparent Power'}
	MDP5001_341_L3_Power_Apparent_Power			AT%I* : REAL;		// linked via attribute 
	{attribute 'TcLinkTo' := 'TIID^Device 2 (EtherCAT)^Term 1 (EK1200)^Term 6 (EL3443)^L3 Power^Reactive Power'}
	MDP5001_341_L3_Power_Reactive_Power			AT%I* : REAL;		// linked via attribute 
	{attribute 'TcLinkTo' := 'TIID^Device 2 (EtherCAT)^Term 1 (EK1200)^Term 6 (EL3443)^L3 Power^Power Factor'}
	MDP5001_341_L3_Power_Power_Factor			AT%I* : REAL;		// linked via attribute 
	{attribute 'TcLinkTo' := 'TIID^Device 2 (EtherCAT)^Term 1 (EK1200)^Term 6 (EL3443)^Total Status^System State'}
	MDP5001_341_Total_Status_System_State				AT%I* : BOOL;		// linked via attribute 
	{attribute 'TcLinkTo' := 'TIID^Device 2 (EtherCAT)^Term 1 (EK1200)^Term 6 (EL3443)^Total Status^Grid Direction'}
	MDP5001_341_Total_Status_Grid_Direction				AT%I* : BOOL;		// linked via attribute 
	{attribute 'TcLinkTo' := 'TIID^Device 2 (EtherCAT)^Term 1 (EK1200)^Term 6 (EL3443)^Total Status^Frequency Guard Warning'}
	MDP5001_341_Total_Status_Frequency_Guard_Warning	AT%I* : BOOL;		// linked via attribute 
	{attribute 'TcLinkTo' := 'TIID^Device 2 (EtherCAT)^Term 1 (EK1200)^Term 6 (EL3443)^Total Status^Frequency Guard Error'}
	MDP5001_341_Total_Status_Frequency_Guard_Error		AT%I* : BOOL;		// linked via attribute 
	{attribute 'TcLinkTo' := 'TIID^Device 2 (EtherCAT)^Term 1 (EK1200)^Term 6 (EL3443)^Total Status^Neutral Current Guard Warning'}
	MDP5001_341_Total_Status_Neutral_Current_Guard_Warning	AT%I* : BOOL;		// linked via attribute 
	{attribute 'TcLinkTo' := 'TIID^Device 2 (EtherCAT)^Term 1 (EK1200)^Term 6 (EL3443)^Total Status^Neutral Current Guard Error'}
	MDP5001_341_Total_Status_Neutral_Current_Guard_Error	AT%I* : BOOL;		// linked via attribute 
	{attribute 'TcLinkTo' := 'TIID^Device 2 (EtherCAT)^Term 1 (EK1200)^Term 6 (EL3443)^Total Status^Active Power Guard Warning'}
	MDP5001_341_Total_Status_Active_Power_Guard_Warning		AT%I* : BOOL;		// linked via attribute 
	{attribute 'TcLinkTo' := 'TIID^Device 2 (EtherCAT)^Term 1 (EK1200)^Term 6 (EL3443)^Total Status^Active Power Guard Error'}
	MDP5001_341_Total_Status_Active_Power_Guard_Error		AT%I* : BOOL;		// linked via attribute 
	{attribute 'TcLinkTo' := 'TIID^Device 2 (EtherCAT)^Term 1 (EK1200)^Term 6 (EL3443)^Total Status^Apparent Power Guard Warning'}
	MDP5001_341_Total_Status_Apparent_Power_Guard_Warning	AT%I* : BOOL;		// linked via attribute 
	{attribute 'TcLinkTo' := 'TIID^Device 2 (EtherCAT)^Term 1 (EK1200)^Term 6 (EL3443)^Total Status^Apparent Power Guard Error'}
	MDP5001_341_Total_Status_Apparent_Power_Guard_Error		AT%I* : BOOL;		// linked via attribute 
	{attribute 'TcLinkTo' := 'TIID^Device 2 (EtherCAT)^Term 1 (EK1200)^Term 6 (EL3443)^Total Status^Power Quality Guard Warning'}
	MDP5001_341_Total_Status_Power_Quality_Guard_Warning	AT%I* : BOOL;		// linked via attribute 
	{attribute 'TcLinkTo' := 'TIID^Device 2 (EtherCAT)^Term 1 (EK1200)^Term 6 (EL3443)^Total Status^Power Quality Guard Error'}
	MDP5001_341_Total_Status_Power_Quality_Guard_Error		AT%I* : BOOL;		// linked via attribute 
	{attribute 'TcLinkTo' := 'TIID^Device 2 (EtherCAT)^Term 1 (EK1200)^Term 6 (EL3443)^Total Status^TxPDO State'}
	MDP5001_341_Total_Status_TxPDO_State					AT%I* : BOOL;		// linked via attribute 
	{attribute 'TcLinkTo' := 'TIID^Device 2 (EtherCAT)^Term 1 (EK1200)^Term 6 (EL3443)^Total Status^TxPDO Toggle'}
	MDP5001_341_Total_Status_TxPDO_Toggle					AT%I* : BOOL;		// linked via attribute 
	{attribute 'TcLinkTo' := 'TIID^Device 2 (EtherCAT)^Term 1 (EK1200)^Term 6 (EL3443)^Total Status^Power Quality Factor'}
	MDP5001_341_Total_Status_Power_Quality_Factor			AT%I* : REAL;		// linked via attribute 
	{attribute 'TcLinkTo' := 'TIID^Device 2 (EtherCAT)^Term 1 (EK1200)^Term 6 (EL3443)^Total Basic^Frequency'}
	MDP5001_341_Total_Basic_Frequency						AT%I* : REAL;		// linked via attribute 
	{attribute 'TcLinkTo' := 'TIID^Device 2 (EtherCAT)^Term 1 (EK1200)^Term 6 (EL3443)^Total Basic^Power Factor'}
	MDP5001_341_Total_Basic_Power_Factor					AT%I* : REAL;		// linked via attribute 
	{attribute 'TcLinkTo' := 'TIID^Device 2 (EtherCAT)^Term 1 (EK1200)^Term 6 (EL3443)^Total Basic^Calculated Neutral Line Current'}
	MDP5001_341_Total_Basic_Calculated_Neutral_Line_Current	AT%I* : REAL;		// linked via attribute 
	{attribute 'TcLinkTo' := 'TIID^Device 2 (EtherCAT)^Term 1 (EK1200)^Term 6 (EL3443)^Total Variant Value In^TxPDO Toggle'}
	MDP5001_341_Total_Variant_Value_In_TxPDO_Toggle			AT%I* : BOOL;		// linked via attribute 
	{attribute 'TcLinkTo' := 'TIID^Device 2 (EtherCAT)^Term 1 (EK1200)^Term 6 (EL3443)^Total Variant Value In^Index 1 REAL'}
	MDP5001_341_Total_Variant_Value_In_Index_1_REAL			AT%I* : UINT;		// linked via attribute 
	{attribute 'TcLinkTo' := 'TIID^Device 2 (EtherCAT)^Term 1 (EK1200)^Term 6 (EL3443)^Total Variant Value In^Value 1 REAL'}
	MDP5001_341_Total_Variant_Value_In_Value_1_REAL			AT%I* : REAL;		// linked via attribute 
	{attribute 'TcLinkTo' := 'TIID^Device 2 (EtherCAT)^Term 1 (EK1200)^Term 6 (EL3443)^Total Variant Value In^Index 2 REAL'}
	MDP5001_341_Total_Variant_Value_In_Index_2_REAL			AT%I* : UINT;		// linked via attribute 
	{attribute 'TcLinkTo' := 'TIID^Device 2 (EtherCAT)^Term 1 (EK1200)^Term 6 (EL3443)^Total Variant Value In^Value 2 REAL'}
	MDP5001_341_Total_Variant_Value_In_Value_2_REAL			AT%I* : REAL;		// linked via attribute 
	{attribute 'TcLinkTo' := 'TIID^Device 2 (EtherCAT)^Term 1 (EK1200)^Term 6 (EL3443)^Total Variant Value In^Index 3 REAL'}
	MDP5001_341_Total_Variant_Value_In_Index_3_REAL			AT%I* : UINT;		// linked via attribute 
	{attribute 'TcLinkTo' := 'TIID^Device 2 (EtherCAT)^Term 1 (EK1200)^Term 6 (EL3443)^Total Variant Value In^Value 3 REAL'}
	MDP5001_341_Total_Variant_Value_In_Value_3_REAL			AT%I* : REAL;		// linked via attribute 
	{attribute 'TcLinkTo' := 'TIID^Device 2 (EtherCAT)^Term 1 (EK1200)^Term 6 (EL3443)^Total Variant Value In^Index 4 ULINT'}
	MDP5001_341_Total_Variant_Value_In_Index_4_ULINT		AT%I* : UINT;		// linked via attribute 
	{attribute 'TcLinkTo' := 'TIID^Device 2 (EtherCAT)^Term 1 (EK1200)^Term 6 (EL3443)^Total Variant Value In^Value 4 ULINT'}
	MDP5001_341_Total_Variant_Value_In_Value_4_ULINT		AT%I* : ULINT;	// linked via attribute 
	{attribute 'TcLinkTo' := 'TIID^Device 2 (EtherCAT)^Term 1 (EK1200)^Term 6 (EL3443)^DPM Data^Data 1'}
	MDP5001_341_DPM_Data_Data_1								AT%I* : UDINT;	// linked via attribute 
	{attribute 'TcLinkTo' := 'TIID^Device 2 (EtherCAT)^Term 1 (EK1200)^Term 6 (EL3443)^DPM Data^Data 2'}
	MDP5001_341_DPM_Data_Data_2								AT%I* : UDINT;	// linked via attribute 
	{attribute 'TcLinkTo' := 'TIID^Device 2 (EtherCAT)^Term 1 (EK1200)^Term 6 (EL3443)^DPM Data^Data 3'}
	MDP5001_341_DPM_Data_Data_3								AT%I* : UDINT;	// linked via attribute 
	{attribute 'TcLinkTo' := 'TIID^Device 2 (EtherCAT)^Term 1 (EK1200)^Term 6 (EL3443)^DPM Data^Data 4'}
	MDP5001_341_DPM_Data_Data_4								AT%I* : UDINT;	// linked via attribute 
	{attribute 'TcLinkTo' := 'TIID^Device 2 (EtherCAT)^Term 1 (EK1200)^Term 6 (EL3443)^DPM Data^Data 5'}
	MDP5001_341_DPM_Data_Data_5								AT%I* : UDINT;	// linked via attribute 
	{attribute 'TcLinkTo' := 'TIID^Device 2 (EtherCAT)^Term 1 (EK1200)^Term 6 (EL3443)^DPM Data^Data 6'}
	MDP5001_341_DPM_Data_Data_6								AT%I* : UDINT;	// linked via attribute 
	{attribute 'TcLinkTo' := 'TIID^Device 2 (EtherCAT)^Term 1 (EK1200)^Term 6 (EL3443)^DPM Data^Data 7'}
	MDP5001_341_DPM_Data_Data_7								AT%I* : UDINT;	// linked via attribute 
	{attribute 'TcLinkTo' := 'TIID^Device 2 (EtherCAT)^Term 1 (EK1200)^Term 6 (EL3443)^DPM Data^Data 8'}
	MDP5001_341_DPM_Data_Data_8								AT%I* : UDINT;	// linked via attribute 
	{attribute 'TcLinkTo' := 'TIID^Device 2 (EtherCAT)^Term 1 (EK1200)^Term 6 (EL3443)^DPM Data^Data 9'}
	MDP5001_341_DPM_Data_Data_9								AT%I* : UDINT;	// linked via attribute 
	{attribute 'TcLinkTo' := 'TIID^Device 2 (EtherCAT)^Term 1 (EK1200)^Term 6 (EL3443)^DPM Data^Data 10'}
	MDP5001_341_DPM_Data_Data_10							AT%I* : UDINT;	// linked via attribute 
	{attribute 'TcLinkTo' := 'TIID^Device 2 (EtherCAT)^Term 1 (EK1200)^Term 6 (EL3443)^DPM Data^Data 11'}
	MDP5001_341_DPM_Data_Data_11							AT%I* : UDINT;	// linked via attribute 
	{attribute 'TcLinkTo' := 'TIID^Device 2 (EtherCAT)^Term 1 (EK1200)^Term 6 (EL3443)^DPM Data^Data 12'}
	MDP5001_341_DPM_Data_Data_12							AT%I* : UDINT;	// linked via attribute 
	{attribute 'TcLinkTo' := 'TIID^Device 2 (EtherCAT)^Term 1 (EK1200)^Term 6 (EL3443)^DPM Data^Data 13'}
	MDP5001_341_DPM_Data_Data_13							AT%I* : UDINT;	// linked via attribute 
	{attribute 'TcLinkTo' := 'TIID^Device 2 (EtherCAT)^Term 1 (EK1200)^Term 6 (EL3443)^DPM Data^Data 14'}
	MDP5001_341_DPM_Data_Data_14							AT%I* : UDINT;	// linked via attribute 
	{attribute 'TcLinkTo' := 'TIID^Device 2 (EtherCAT)^Term 1 (EK1200)^Term 6 (EL3443)^DPM Data^Data 15'}
	MDP5001_341_DPM_Data_Data_15							AT%I* : UDINT;	// linked via attribute 
	{attribute 'TcLinkTo' := 'TIID^Device 2 (EtherCAT)^Term 1 (EK1200)^Term 6 (EL3443)^DPM Data^Data 16'}
	MDP5001_341_DPM_Data_Data_16							AT%I* : UDINT;	// linked via attribute 
	{attribute 'TcLinkTo' := 'TIID^Device 2 (EtherCAT)^Term 1 (EK1200)^Term 6 (EL3443)^DPM Data^Data 17'}
	MDP5001_341_DPM_Data_Data_17							AT%I* : UDINT;	// linked via attribute 
	{attribute 'TcLinkTo' := 'TIID^Device 2 (EtherCAT)^Term 1 (EK1200)^Term 6 (EL3443)^DPM Data^Data 18'}
	MDP5001_341_DPM_Data_Data_18							AT%I* : UDINT;	// linked via attribute 
	{attribute 'TcLinkTo' := 'TIID^Device 2 (EtherCAT)^Term 1 (EK1200)^Term 6 (EL3443)^DPM Data^Data 19'}
	MDP5001_341_DPM_Data_Data_19							AT%I* : UDINT;	// linked via attribute 
	{attribute 'TcLinkTo' := 'TIID^Device 2 (EtherCAT)^Term 1 (EK1200)^Term 6 (EL3443)^DPM Data^Data 20'}
	MDP5001_341_DPM_Data_Data_20							AT%I* : UDINT;	// linked via attribute 
	{attribute 'TcLinkTo' := 'TIID^Device 2 (EtherCAT)^Term 1 (EK1200)^Term 6 (EL3443)^Total Variant Value Out^Index 1 REAL'}
	MDP5001_341_Total_Variant_Value_Out_Index_1_REAL	AT%Q* : UINT;
	{attribute 'TcLinkTo' := 'TIID^Device 2 (EtherCAT)^Term 1 (EK1200)^Term 6 (EL3443)^Total Variant Value Out^Index 2 REAL'}
	MDP5001_341_Total_Variant_Value_Out_Index_2_REAL	AT%Q* : UINT;
	{attribute 'TcLinkTo' := 'TIID^Device 2 (EtherCAT)^Term 1 (EK1200)^Term 6 (EL3443)^Total Variant Value Out^Index 3 REAL'}
	MDP5001_341_Total_Variant_Value_Out_Index_3_REAL	AT%Q* : UINT;
	{attribute 'TcLinkTo' := 'TIID^Device 2 (EtherCAT)^Term 1 (EK1200)^Term 6 (EL3443)^Total Variant Value Out^Index 4 ULINT'}
	MDP5001_341_Total_Variant_Value_Out_Index_4_ULINT	AT%Q* : UINT;
	{attribute 'TcLinkTo' := 'TIID^Device 2 (EtherCAT)^Term 1 (EK1200)^Term 6 (EL3443)^Total Interval^Reset Interval'}
	MDP5001_341_Total_Interval_Reset_Interval			AT%Q* : BOOL;	

	// IOs for EL3443
	{attribute 'TcLinkTo' := 'TIID^Device 2 (EtherCAT)^Term 1 (EK1200)^Term 2 (EL3443)^L1 Status^Voltage Sign Bit'}
	MDP5001_342_L1_Status_Voltage_Sign_Bit   	AT%I*  : BOOL;  // linked via attribute 
	{attribute 'TcLinkTo' := 'TIID^Device 2 (EtherCAT)^Term 1 (EK1200)^Term 2 (EL3443)^L1 Status^Overvoltage'}
	MDP5001_342_L1_Status_Overvoltage			AT%I*  : BOOL;  // linked via attribute 
	{attribute 'TcLinkTo' := 'TIID^Device 2 (EtherCAT)^Term 1 (EK1200)^Term 2 (EL3443)^L1 Status^Overcurrent'}
	MDP5001_342_L1_Status_Overcurrent			AT%I*  : BOOL;  // linked via attribute 
	{attribute 'TcLinkTo' := 'TIID^Device 2 (EtherCAT)^Term 1 (EK1200)^Term 2 (EL3443)^L1 Status^Inaccurate Voltage'}	
	MDP5001_342_L1_Status_Inaccurate_Voltage	AT%I*  : BOOL;  // linked via attribute 
	{attribute 'TcLinkTo' := 'TIID^Device 2 (EtherCAT)^Term 1 (EK1200)^Term 2 (EL3443)^L1 Status^Inaccurate Current'}
	MDP5001_342_L1_Status_Inaccurate_Current	AT%I*  : BOOL;  // linked via attribute 	
	{attribute 'TcLinkTo' := 'TIID^Device 2 (EtherCAT)^Term 1 (EK1200)^Term 2 (EL3443)^L1 Status^Voltage Guard Warning'}
	MDP5001_342_L1_Status_Voltage_Guard_Warning	AT%I*  : BOOL;  // linked via attribute
	{attribute 'TcLinkTo' := 'TIID^Device 2 (EtherCAT)^Term 1 (EK1200)^Term 2 (EL3443)^L1 Status^Voltage Guard Error'}
	MDP5001_342_L1_Status_Voltage_Guard_Error	AT%I*  : BOOL;  // linked via attribute
	{attribute 'TcLinkTo' := 'TIID^Device 2 (EtherCAT)^Term 1 (EK1200)^Term 2 (EL3443)^L1 Status^Current Guard Warning'}
	MDP5001_342_L1_Status_Current_Guard_Warning AT%I*  : BOOL;  // linked via attribute
	{attribute 'TcLinkTo' := 'TIID^Device 2 (EtherCAT)^Term 1 (EK1200)^Term 2 (EL3443)^L1 Status^Current Guard Error'}
	MDP5001_342_L1_Status_Current_Guard_Error	AT%I*  : BOOL;  // linked via attribute
	{attribute 'TcLinkTo' := 'TIID^Device 2 (EtherCAT)^Term 1 (EK1200)^Term 2 (EL3443)^L1 Status^TxPDO Toggle'}
	MDP5001_342_L1_Status_TxPDO_Toggle			AT%I*  : BOOL;  // linked via attribute
	{attribute 'TcLinkTo' := 'TIID^Device 2 (EtherCAT)^Term 1 (EK1200)^Term 2 (EL3443)^L1 Basic^Voltage'}
	MDP5001_342_L1_Basic_Voltage				AT%I*  : REAL;		// linked via attribute 
	{attribute 'TcLinkTo' := 'TIID^Device 2 (EtherCAT)^Term 1 (EK1200)^Term 2 (EL3443)^L1 Basic^Current'}
	MDP5001_342_L1_Basic_Current				AT%I*  : REAL;		// linked via attribute 
	{attribute 'TcLinkTo' := 'TIID^Device 2 (EtherCAT)^Term 1 (EK1200)^Term 2 (EL3443)^L1 Power^Active Power'}
	MDP5001_342_L1_Power_Active_Power			AT%I*  : REAL;		// linked via attribute 
	{attribute 'TcLinkTo' := 'TIID^Device 2 (EtherCAT)^Term 1 (EK1200)^Term 2 (EL3443)^L1 Power^Apparent Power'}
	MDP5001_342_L1_Power_Apparent_Power			AT%I* : REAL;		// linked via attribute 
	{attribute 'TcLinkTo' := 'TIID^Device 2 (EtherCAT)^Term 1 (EK1200)^Term 2 (EL3443)^L1 Power^Reactive Power'}
	MDP5001_342_L1_Power_Reactive_Power			AT%I* : REAL;		// linked via attribute 
	{attribute 'TcLinkTo' := 'TIID^Device 2 (EtherCAT)^Term 1 (EK1200)^Term 2 (EL3443)^L1 Power^Power Factor'}
	MDP5001_342_L1_Power_Power_Factor			AT%I* : REAL;		// linked via attribute 
	{attribute 'TcLinkTo' := 'TIID^Device 2 (EtherCAT)^Term 1 (EK1200)^Term 2 (EL3443)^L2 Status^Voltage Sign Bit'}
	MDP5001_342_L2_Status_Voltage_Sign_Bit   	AT%I*  : BOOL;  // linked via attribute 
	{attribute 'TcLinkTo' := 'TIID^Device 2 (EtherCAT)^Term 1 (EK1200)^Term 2 (EL3443)^L2 Status^Overvoltage'}
	MDP5001_342_L2_Status_Overvoltage			AT%I*  : BOOL;  // linked via attribute 
	{attribute 'TcLinkTo' := 'TIID^Device 2 (EtherCAT)^Term 1 (EK1200)^Term 2 (EL3443)^L2 Status^Overcurrent'}
	MDP5001_342_L2_Status_Overcurrent			AT%I*  : BOOL;  // linked via attribute 
	{attribute 'TcLinkTo' := 'TIID^Device 2 (EtherCAT)^Term 1 (EK1200)^Term 2 (EL3443)^L2 Status^Inaccurate Voltage'}	
	MDP5001_342_L2_Status_Inaccurate_Voltage	AT%I*  : BOOL;  // linked via attribute 
	{attribute 'TcLinkTo' := 'TIID^Device 2 (EtherCAT)^Term 1 (EK1200)^Term 2 (EL3443)^L2 Status^Inaccurate Current'}
	MDP5001_342_L2_Status_Inaccurate_Current	AT%I*  : BOOL;  // linked via attribute 	
	{attribute 'TcLinkTo' := 'TIID^Device 2 (EtherCAT)^Term 1 (EK1200)^Term 2 (EL3443)^L2 Status^Voltage Guard Warning'}
	MDP5001_342_L2_Status_Voltage_Guard_Warning	AT%I*  : BOOL;  // linked via attribute
	{attribute 'TcLinkTo' := 'TIID^Device 2 (EtherCAT)^Term 1 (EK1200)^Term 2 (EL3443)^L2 Status^Voltage Guard Error'}
	MDP5001_342_L2_Status_Voltage_Guard_Error	AT%I*  : BOOL;  // linked via attribute
	{attribute 'TcLinkTo' := 'TIID^Device 2 (EtherCAT)^Term 1 (EK1200)^Term 2 (EL3443)^L2 Status^Current Guard Warning'}
	MDP5001_342_L2_Status_Current_Guard_Warning AT%I*  : BOOL;  // linked via attribute
	{attribute 'TcLinkTo' := 'TIID^Device 2 (EtherCAT)^Term 1 (EK1200)^Term 2 (EL3443)^L2 Status^Current Guard Error'}
	MDP5001_342_L2_Status_Current_Guard_Error	AT%I*  : BOOL;  // linked via attribute
	{attribute 'TcLinkTo' := 'TIID^Device 2 (EtherCAT)^Term 1 (EK1200)^Term 2 (EL3443)^L2 Status^TxPDO Toggle'}
	MDP5001_342_L2_Status_TxPDO_Toggle			AT%I*  : BOOL;  // linked via attribute
	{attribute 'TcLinkTo' := 'TIID^Device 2 (EtherCAT)^Term 1 (EK1200)^Term 2 (EL3443)^L2 Basic^Voltage'}
	MDP5001_342_L2_Basic_Voltage				AT%I* : REAL;		// linked via attribute 
	{attribute 'TcLinkTo' := 'TIID^Device 2 (EtherCAT)^Term 1 (EK1200)^Term 2 (EL3443)^L2 Basic^Current'}
	MDP5001_342_L2_Basic_Current				AT%I* : REAL;		// linked via attribute 
	{attribute 'TcLinkTo' := 'TIID^Device 2 (EtherCAT)^Term 1 (EK1200)^Term 2 (EL3443)^L2 Power^Active Power'}
	MDP5001_342_L2_Power_Active_Power			AT%I* : REAL;		// linked via attribute 
	{attribute 'TcLinkTo' := 'TIID^Device 2 (EtherCAT)^Term 1 (EK1200)^Term 2 (EL3443)^L2 Power^Apparent Power'}
	MDP5001_342_L2_Power_Apparent_Power			AT%I* : REAL;		// linked via attribute 
	{attribute 'TcLinkTo' := 'TIID^Device 2 (EtherCAT)^Term 1 (EK1200)^Term 2 (EL3443)^L2 Power^Reactive Power'}
	MDP5001_342_L2_Power_Reactive_Power			AT%I* : REAL;		// linked via attribute 
	{attribute 'TcLinkTo' := 'TIID^Device 2 (EtherCAT)^Term 1 (EK1200)^Term 2 (EL3443)^L2 Power^Power Factor'}
	MDP5001_342_L2_Power_Power_Factor			AT%I* : REAL;		// linked via attribute 
	{attribute 'TcLinkTo' := 'TIID^Device 2 (EtherCAT)^Term 1 (EK1200)^Term 2 (EL3443)^L3 Status^Voltage Sign Bit'}
	MDP5001_342_L3_Status_Voltage_Sign_Bit   	AT%I*  : BOOL;  // linked via attribute 
	{attribute 'TcLinkTo' := 'TIID^Device 2 (EtherCAT)^Term 1 (EK1200)^Term 2 (EL3443)^L3 Status^Overvoltage'}
	MDP5001_342_L3_Status_Overvoltage			AT%I*  : BOOL;  // linked via attribute 
	{attribute 'TcLinkTo' := 'TIID^Device 2 (EtherCAT)^Term 1 (EK1200)^Term 2 (EL3443)^L3 Status^Overcurrent'}
	MDP5001_342_L3_Status_Overcurrent			AT%I*  : BOOL;  // linked via attribute 
	{attribute 'TcLinkTo' := 'TIID^Device 2 (EtherCAT)^Term 1 (EK1200)^Term 2 (EL3443)^L3 Status^Inaccurate Voltage'}	
	MDP5001_342_L3_Status_Inaccurate_Voltage	AT%I*  : BOOL;  // linked via attribute 
	{attribute 'TcLinkTo' := 'TIID^Device 2 (EtherCAT)^Term 1 (EK1200)^Term 2 (EL3443)^L3 Status^Inaccurate Current'}
	MDP5001_342_L3_Status_Inaccurate_Current	AT%I*  : BOOL;  // linked via attribute 	
	{attribute 'TcLinkTo' := 'TIID^Device 2 (EtherCAT)^Term 1 (EK1200)^Term 2 (EL3443)^L3 Status^Voltage Guard Warning'}
	MDP5001_342_L3_Status_Voltage_Guard_Warning	AT%I*  : BOOL;  // linked via attribute
	{attribute 'TcLinkTo' := 'TIID^Device 2 (EtherCAT)^Term 1 (EK1200)^Term 2 (EL3443)^L3 Status^Voltage Guard Error'}
	MDP5001_342_L3_Status_Voltage_Guard_Error	AT%I*  : BOOL;  // linked via attribute
	{attribute 'TcLinkTo' := 'TIID^Device 2 (EtherCAT)^Term 1 (EK1200)^Term 2 (EL3443)^L3 Status^Current Guard Warning'}
	MDP5001_342_L3_Status_Current_Guard_Warning AT%I*  : BOOL;  // linked via attribute
	{attribute 'TcLinkTo' := 'TIID^Device 2 (EtherCAT)^Term 1 (EK1200)^Term 2 (EL3443)^L3 Status^Current Guard Error'}
	MDP5001_342_L3_Status_Current_Guard_Error	AT%I*  : BOOL;  // linked via attribute
	{attribute 'TcLinkTo' := 'TIID^Device 2 (EtherCAT)^Term 1 (EK1200)^Term 2 (EL3443)^L3 Status^TxPDO Toggle'}
	MDP5001_342_L3_Status_TxPDO_Toggle			AT%I*  : BOOL;  // linked via attribute
	{attribute 'TcLinkTo' := 'TIID^Device 2 (EtherCAT)^Term 1 (EK1200)^Term 2 (EL3443)^L3 Basic^Voltage'}
	MDP5001_342_L3_Basic_Voltage				AT%I* : REAL;		// linked via attribute 
	{attribute 'TcLinkTo' := 'TIID^Device 2 (EtherCAT)^Term 1 (EK1200)^Term 2 (EL3443)^L3 Basic^Current'}
	MDP5001_342_L3_Basic_Current				AT%I* : REAL;		// linked via attribute 
	{attribute 'TcLinkTo' := 'TIID^Device 2 (EtherCAT)^Term 1 (EK1200)^Term 2 (EL3443)^L3 Power^Active Power'}
	MDP5001_342_L3_Power_Active_Power			AT%I* : REAL;		// linked via attribute 
	{attribute 'TcLinkTo' := 'TIID^Device 2 (EtherCAT)^Term 1 (EK1200)^Term 2 (EL3443)^L3 Power^Apparent Power'}
	MDP5001_342_L3_Power_Apparent_Power			AT%I* : REAL;		// linked via attribute 
	{attribute 'TcLinkTo' := 'TIID^Device 2 (EtherCAT)^Term 1 (EK1200)^Term 2 (EL3443)^L3 Power^Reactive Power'}
	MDP5001_342_L3_Power_Reactive_Power			AT%I* : REAL;		// linked via attribute 
	{attribute 'TcLinkTo' := 'TIID^Device 2 (EtherCAT)^Term 1 (EK1200)^Term 2 (EL3443)^L3 Power^Power Factor'}
	MDP5001_342_L3_Power_Power_Factor			AT%I* : REAL;		// linked via attribute 
	{attribute 'TcLinkTo' := 'TIID^Device 2 (EtherCAT)^Term 1 (EK1200)^Term 2 (EL3443)^Total Status^System State'}
	MDP5001_342_Total_Status_System_State				AT%I* : BOOL;		// linked via attribute 
	{attribute 'TcLinkTo' := 'TIID^Device 2 (EtherCAT)^Term 1 (EK1200)^Term 2 (EL3443)^Total Status^Grid Direction'}
	MDP5001_342_Total_Status_Grid_Direction				AT%I* : BOOL;		// linked via attribute 
	{attribute 'TcLinkTo' := 'TIID^Device 2 (EtherCAT)^Term 1 (EK1200)^Term 2 (EL3443)^Total Status^Frequency Guard Warning'}
	MDP5001_342_Total_Status_Frequency_Guard_Warning	AT%I* : BOOL;		// linked via attribute 
	{attribute 'TcLinkTo' := 'TIID^Device 2 (EtherCAT)^Term 1 (EK1200)^Term 2 (EL3443)^Total Status^Frequency Guard Error'}
	MDP5001_342_Total_Status_Frequency_Guard_Error		AT%I* : BOOL;		// linked via attribute 
	{attribute 'TcLinkTo' := 'TIID^Device 2 (EtherCAT)^Term 1 (EK1200)^Term 2 (EL3443)^Total Status^Neutral Current Guard Warning'}
	MDP5001_342_Total_Status_Neutral_Current_Guard_Warning	AT%I* : BOOL;		// linked via attribute 
	{attribute 'TcLinkTo' := 'TIID^Device 2 (EtherCAT)^Term 1 (EK1200)^Term 2 (EL3443)^Total Status^Neutral Current Guard Error'}
	MDP5001_342_Total_Status_Neutral_Current_Guard_Error	AT%I* : BOOL;		// linked via attribute 
	{attribute 'TcLinkTo' := 'TIID^Device 2 (EtherCAT)^Term 1 (EK1200)^Term 2 (EL3443)^Total Status^Active Power Guard Warning'}
	MDP5001_342_Total_Status_Active_Power_Guard_Warning		AT%I* : BOOL;		// linked via attribute 
	{attribute 'TcLinkTo' := 'TIID^Device 2 (EtherCAT)^Term 1 (EK1200)^Term 2 (EL3443)^Total Status^Active Power Guard Error'}
	MDP5001_342_Total_Status_Active_Power_Guard_Error		AT%I* : BOOL;		// linked via attribute 
	{attribute 'TcLinkTo' := 'TIID^Device 2 (EtherCAT)^Term 1 (EK1200)^Term 2 (EL3443)^Total Status^Apparent Power Guard Warning'}
	MDP5001_342_Total_Status_Apparent_Power_Guard_Warning	AT%I* : BOOL;		// linked via attribute 
	{attribute 'TcLinkTo' := 'TIID^Device 2 (EtherCAT)^Term 1 (EK1200)^Term 2 (EL3443)^Total Status^Apparent Power Guard Error'}
	MDP5001_342_Total_Status_Apparent_Power_Guard_Error		AT%I* : BOOL;		// linked via attribute 
	{attribute 'TcLinkTo' := 'TIID^Device 2 (EtherCAT)^Term 1 (EK1200)^Term 2 (EL3443)^Total Status^Power Quality Guard Warning'}
	MDP5001_342_Total_Status_Power_Quality_Guard_Warning	AT%I* : BOOL;		// linked via attribute 
	{attribute 'TcLinkTo' := 'TIID^Device 2 (EtherCAT)^Term 1 (EK1200)^Term 2 (EL3443)^Total Status^Power Quality Guard Error'}
	MDP5001_342_Total_Status_Power_Quality_Guard_Error		AT%I* : BOOL;		// linked via attribute 
	{attribute 'TcLinkTo' := 'TIID^Device 2 (EtherCAT)^Term 1 (EK1200)^Term 2 (EL3443)^Total Status^TxPDO State'}
	MDP5001_342_Total_Status_TxPDO_State					AT%I* : BOOL;		// linked via attribute 
	{attribute 'TcLinkTo' := 'TIID^Device 2 (EtherCAT)^Term 1 (EK1200)^Term 2 (EL3443)^Total Status^TxPDO Toggle'}
	MDP5001_342_Total_Status_TxPDO_Toggle					AT%I* : BOOL;		// linked via attribute 
	{attribute 'TcLinkTo' := 'TIID^Device 2 (EtherCAT)^Term 1 (EK1200)^Term 2 (EL3443)^Total Status^Power Quality Factor'}
	MDP5001_342_Total_Status_Power_Quality_Factor			AT%I* : REAL;		// linked via attribute 
	{attribute 'TcLinkTo' := 'TIID^Device 2 (EtherCAT)^Term 1 (EK1200)^Term 2 (EL3443)^Total Basic^Frequency'}
	MDP5001_342_Total_Basic_Frequency						AT%I* : REAL;		// linked via attribute 
	{attribute 'TcLinkTo' := 'TIID^Device 2 (EtherCAT)^Term 1 (EK1200)^Term 2 (EL3443)^Total Basic^Power Factor'}
	MDP5001_342_Total_Basic_Power_Factor					AT%I* : REAL;		// linked via attribute 
	{attribute 'TcLinkTo' := 'TIID^Device 2 (EtherCAT)^Term 1 (EK1200)^Term 2 (EL3443)^Total Basic^Calculated Neutral Line Current'}
	MDP5001_342_Total_Basic_Calculated_Neutral_Line_Current	AT%I* : REAL;		// linked via attribute 
	{attribute 'TcLinkTo' := 'TIID^Device 2 (EtherCAT)^Term 1 (EK1200)^Term 2 (EL3443)^Total Variant Value In^TxPDO Toggle'}
	MDP5001_342_Total_Variant_Value_In_TxPDO_Toggle			AT%I* : BOOL;		// linked via attribute 
	{attribute 'TcLinkTo' := 'TIID^Device 2 (EtherCAT)^Term 1 (EK1200)^Term 2 (EL3443)^Total Variant Value In^Index 1 REAL'}
	MDP5001_342_Total_Variant_Value_In_Index_1_REAL			AT%I* : UINT;		// linked via attribute 
	{attribute 'TcLinkTo' := 'TIID^Device 2 (EtherCAT)^Term 1 (EK1200)^Term 2 (EL3443)^Total Variant Value In^Value 1 REAL'}
	MDP5001_342_Total_Variant_Value_In_Value_1_REAL			AT%I* : REAL;		// linked via attribute 
	{attribute 'TcLinkTo' := 'TIID^Device 2 (EtherCAT)^Term 1 (EK1200)^Term 2 (EL3443)^Total Variant Value In^Index 2 REAL'}
	MDP5001_342_Total_Variant_Value_In_Index_2_REAL			AT%I* : UINT;		// linked via attribute 
	{attribute 'TcLinkTo' := 'TIID^Device 2 (EtherCAT)^Term 1 (EK1200)^Term 2 (EL3443)^Total Variant Value In^Value 2 REAL'}
	MDP5001_342_Total_Variant_Value_In_Value_2_REAL			AT%I* : REAL;		// linked via attribute 
	{attribute 'TcLinkTo' := 'TIID^Device 2 (EtherCAT)^Term 1 (EK1200)^Term 2 (EL3443)^Total Variant Value In^Index 3 REAL'}
	MDP5001_342_Total_Variant_Value_In_Index_3_REAL			AT%I* : UINT;		// linked via attribute 
	{attribute 'TcLinkTo' := 'TIID^Device 2 (EtherCAT)^Term 1 (EK1200)^Term 2 (EL3443)^Total Variant Value In^Value 3 REAL'}
	MDP5001_342_Total_Variant_Value_In_Value_3_REAL			AT%I* : REAL;		// linked via attribute 
	{attribute 'TcLinkTo' := 'TIID^Device 2 (EtherCAT)^Term 1 (EK1200)^Term 2 (EL3443)^Total Variant Value In^Index 4 ULINT'}
	MDP5001_342_Total_Variant_Value_In_Index_4_ULINT		AT%I* : UINT;		// linked via attribute 
	{attribute 'TcLinkTo' := 'TIID^Device 2 (EtherCAT)^Term 1 (EK1200)^Term 2 (EL3443)^Total Variant Value In^Value 4 ULINT'}
	MDP5001_342_Total_Variant_Value_In_Value_4_ULINT		AT%I* : ULINT;	// linked via attribute 
	{attribute 'TcLinkTo' := 'TIID^Device 2 (EtherCAT)^Term 1 (EK1200)^Term 2 (EL3443)^DPM Data^Data 1'}
	MDP5001_342_DPM_Data_Data_1								AT%I* : UDINT;	// linked via attribute 
	{attribute 'TcLinkTo' := 'TIID^Device 2 (EtherCAT)^Term 1 (EK1200)^Term 2 (EL3443)^DPM Data^Data 2'}
	MDP5001_342_DPM_Data_Data_2								AT%I* : UDINT;	// linked via attribute 
	{attribute 'TcLinkTo' := 'TIID^Device 2 (EtherCAT)^Term 1 (EK1200)^Term 2 (EL3443)^DPM Data^Data 3'}
	MDP5001_342_DPM_Data_Data_3								AT%I* : UDINT;	// linked via attribute 
	{attribute 'TcLinkTo' := 'TIID^Device 2 (EtherCAT)^Term 1 (EK1200)^Term 2 (EL3443)^DPM Data^Data 4'}
	MDP5001_342_DPM_Data_Data_4								AT%I* : UDINT;	// linked via attribute 
	{attribute 'TcLinkTo' := 'TIID^Device 2 (EtherCAT)^Term 1 (EK1200)^Term 2 (EL3443)^DPM Data^Data 5'}
	MDP5001_342_DPM_Data_Data_5								AT%I* : UDINT;	// linked via attribute 
	{attribute 'TcLinkTo' := 'TIID^Device 2 (EtherCAT)^Term 1 (EK1200)^Term 2 (EL3443)^DPM Data^Data 6'}
	MDP5001_342_DPM_Data_Data_6								AT%I* : UDINT;	// linked via attribute 
	{attribute 'TcLinkTo' := 'TIID^Device 2 (EtherCAT)^Term 1 (EK1200)^Term 2 (EL3443)^DPM Data^Data 7'}
	MDP5001_342_DPM_Data_Data_7								AT%I* : UDINT;	// linked via attribute 
	{attribute 'TcLinkTo' := 'TIID^Device 2 (EtherCAT)^Term 1 (EK1200)^Term 2 (EL3443)^DPM Data^Data 8'}
	MDP5001_342_DPM_Data_Data_8								AT%I* : UDINT;	// linked via attribute 
	{attribute 'TcLinkTo' := 'TIID^Device 2 (EtherCAT)^Term 1 (EK1200)^Term 2 (EL3443)^DPM Data^Data 9'}
	MDP5001_342_DPM_Data_Data_9								AT%I* : UDINT;	// linked via attribute 
	{attribute 'TcLinkTo' := 'TIID^Device 2 (EtherCAT)^Term 1 (EK1200)^Term 2 (EL3443)^DPM Data^Data 10'}
	MDP5001_342_DPM_Data_Data_10							AT%I* : UDINT;	// linked via attribute 
	{attribute 'TcLinkTo' := 'TIID^Device 2 (EtherCAT)^Term 1 (EK1200)^Term 2 (EL3443)^DPM Data^Data 11'}
	MDP5001_342_DPM_Data_Data_11							AT%I* : UDINT;	// linked via attribute 
	{attribute 'TcLinkTo' := 'TIID^Device 2 (EtherCAT)^Term 1 (EK1200)^Term 2 (EL3443)^DPM Data^Data 12'}
	MDP5001_342_DPM_Data_Data_12							AT%I* : UDINT;	// linked via attribute 
	{attribute 'TcLinkTo' := 'TIID^Device 2 (EtherCAT)^Term 1 (EK1200)^Term 2 (EL3443)^DPM Data^Data 13'}
	MDP5001_342_DPM_Data_Data_13							AT%I* : UDINT;	// linked via attribute 
	{attribute 'TcLinkTo' := 'TIID^Device 2 (EtherCAT)^Term 1 (EK1200)^Term 2 (EL3443)^DPM Data^Data 14'}
	MDP5001_342_DPM_Data_Data_14							AT%I* : UDINT;	// linked via attribute 
	{attribute 'TcLinkTo' := 'TIID^Device 2 (EtherCAT)^Term 1 (EK1200)^Term 2 (EL3443)^DPM Data^Data 15'}
	MDP5001_342_DPM_Data_Data_15							AT%I* : UDINT;	// linked via attribute 
	{attribute 'TcLinkTo' := 'TIID^Device 2 (EtherCAT)^Term 1 (EK1200)^Term 2 (EL3443)^DPM Data^Data 16'}
	MDP5001_342_DPM_Data_Data_16							AT%I* : UDINT;	// linked via attribute 
	{attribute 'TcLinkTo' := 'TIID^Device 2 (EtherCAT)^Term 1 (EK1200)^Term 2 (EL3443)^DPM Data^Data 17'}
	MDP5001_342_DPM_Data_Data_17							AT%I* : UDINT;	// linked via attribute 
	{attribute 'TcLinkTo' := 'TIID^Device 2 (EtherCAT)^Term 1 (EK1200)^Term 2 (EL3443)^DPM Data^Data 18'}
	MDP5001_342_DPM_Data_Data_18							AT%I* : UDINT;	// linked via attribute 
	{attribute 'TcLinkTo' := 'TIID^Device 2 (EtherCAT)^Term 1 (EK1200)^Term 2 (EL3443)^DPM Data^Data 19'}
	MDP5001_342_DPM_Data_Data_19							AT%I* : UDINT;	// linked via attribute 
	{attribute 'TcLinkTo' := 'TIID^Device 2 (EtherCAT)^Term 1 (EK1200)^Term 2 (EL3443)^DPM Data^Data 20'}
	MDP5001_342_DPM_Data_Data_20							AT%I* : UDINT;	// linked via attribute 
	{attribute 'TcLinkTo' := 'TIID^Device 2 (EtherCAT)^Term 1 (EK1200)^Term 2 (EL3443)^Total Variant Value Out^Index 1 REAL'}
	MDP5001_342_Total_Variant_Value_Out_Index_1_REAL	AT%Q* : UINT;
	{attribute 'TcLinkTo' := 'TIID^Device 2 (EtherCAT)^Term 1 (EK1200)^Term 2 (EL3443)^Total Variant Value Out^Index 2 REAL'}
	MDP5001_342_Total_Variant_Value_Out_Index_2_REAL	AT%Q* : UINT;
	{attribute 'TcLinkTo' := 'TIID^Device 2 (EtherCAT)^Term 1 (EK1200)^Term 2 (EL3443)^Total Variant Value Out^Index 3 REAL'}
	MDP5001_342_Total_Variant_Value_Out_Index_3_REAL	AT%Q* : UINT;
	{attribute 'TcLinkTo' := 'TIID^Device 2 (EtherCAT)^Term 1 (EK1200)^Term 2 (EL3443)^Total Variant Value Out^Index 4 ULINT'}
	MDP5001_342_Total_Variant_Value_Out_Index_4_ULINT	AT%Q* : UINT;
	{attribute 'TcLinkTo' := 'TIID^Device 2 (EtherCAT)^Term 1 (EK1200)^Term 2 (EL3443)^Total Interval^Reset Interval'}
	MDP5001_342_Total_Interval_Reset_Interval			AT%Q* : BOOL;
	
